METHOD PUBLIC Clone : I_Node
VAR
	pNode : POINTER TO LT_INT;
END_VAR
pNode := __NEW(LT_INT);
Clone := pNode^;
END_METHOD

METHOD PROTECTED OnExecute
VAR
END_VAR
out.Value := in1.Value < in2.Value;
END_METHOD

END_FUNCTION_BLOCK

// Comparison/Nodes/LT/LT_LINT
{attribute 'linkalways'} 
{attribute 'no_explicit_call' := 'This FB is a CLASS and must be accessed using methods or properties'}
{attribute 'enable_dynamic_creation'}
FUNCTION_BLOCK FINAL LT_LINT EXTENDS Node
VAR
	in1 : _LINT(0);
	in2 : _LINT(0);
	out : _BOOL(FALSE);
END_VAR

METHOD FB_init : BOOL
VAR_INPUT
	bInitRetains : BOOL; // if TRUE, the retain variables are initialized (warm start / cold start)
	bInCopyCode : BOOL;  // if TRUE, the instance afterwards gets moved into the copy code (online change)
END_VAR
AddInput('in1',THIS^.in1);
AddInput('in2',THIS^.in2);
AddOutput('out', THIS^.out);
END_METHOD

METHOD PUBLIC Clone : I_Node
VAR
	pNode : POINTER TO LT_LINT;
END_VAR
pNode := __NEW(LT_LINT);
Clone := pNode^;
END_METHOD

METHOD PROTECTED OnExecute
VAR
END_VAR
out.Value := in1.Value < in2.Value;
END_METHOD

END_FUNCTION_BLOCK

// Comparison/Nodes/LT/LT_LREAL
{attribute 'linkalways'} 
{attribute 'no_explicit_call' := 'This FB is a CLASS and must be accessed using methods or properties'}
{attribute 'enable_dynamic_creation'}
FUNCTION_BLOCK FINAL LT_LREAL EXTENDS Node
VAR
	in1 : _LREAL(0.0);
	in2 : _LREAL(0.0);
	out : _BOOL(FALSE);
END_VAR

METHOD FB_init : BOOL
VAR_INPUT
	bInitRetains : BOOL; // if TRUE, the retain variables are initialized (warm start / cold start)
	bInCopyCode : BOOL;  // if TRUE, the instance afterwards gets moved into the copy code (online change)
END_VAR
AddInput('in1',THIS^.in1);
AddInput('in2',THIS^.in2);
AddOutput('out', THIS^.out);
END_METHOD

METHOD PUBLIC Clone : I_Node
VAR
	pNode : POINTER TO LT_LREAL;
END_VAR
pNode := __NEW(LT_LREAL);
Clone := pNode^;
END_METHOD

METHOD PROTECTED OnExecute
VAR
END_VAR
out.Value := in1.Value < in2.Value;
END_METHOD

END_FUNCTION_BLOCK

// Comparison/Nodes/LT/LT_LWORD
{attribute 'linkalways'} 
{attribute 'no_explicit_call' := 'This FB is a CLASS and must be accessed using methods or properties'}
{attribute 'enable_dynamic_creation'}
FUNCTION_BLOCK FINAL LT_LWORD EXTENDS Node
VAR
	in1 : _LWORD(0);
	in2 : _LWORD(0);
	out : _BOOL(FALSE);
END_VAR

METHOD FB_init : BOOL
VAR_INPUT
	bInitRetains : BOOL; // if TRUE, the retain variables are initialized (warm start / cold start)
	bInCopyCode : BOOL;  // if TRUE, the instance afterwards gets moved into the copy code (online change)
END_VAR
AddInput('in1',THIS^.in1);
AddInput('in2',THIS^.in2);
AddOutput('out', THIS^.out);
END_METHOD

METHOD PUBLIC Clone : I_Node
VAR
	pNode : POINTER TO LT_LWORD;
END_VAR
pNode := __NEW(LT_LWORD);
Clone := pNode^;
END_METHOD

METHOD PROTECTED OnExecute
VAR
END_VAR
out.Value := in1.Value < in2.Value;
END_METHOD

END_FUNCTION_BLOCK

// Comparison/Nodes/LT/LT_REAL
{attribute 'linkalways'} 
{attribute 'no_explicit_call' := 'This FB is a CLASS and must be accessed using methods or properties'}
{attribute 'enable_dynamic_creation'}
FUNCTION_BLOCK FINAL LT_REAL EXTENDS Node
VAR
	in1 : _REAL(0.0);
	in2 : _REAL(0.0);
	out : _BOOL(FALSE);
END_VAR

METHOD FB_init : BOOL
VAR_INPUT
	bInitRetains : BOOL; // if TRUE, the retain variables are initialized (warm start / cold start)
	bInCopyCode : BOOL;  // if TRUE, the instance afterwards gets moved into the copy code (online change)
END_VAR
AddInput('in1',THIS^.in1);
AddInput('in2',THIS^.in2);
AddOutput('out', THIS^.out);
END_METHOD

METHOD PUBLIC Clone : I_Node
VAR
	pNode : POINTER TO LT_REAL;
END_VAR
pNode := __NEW(LT_REAL);
Clone := pNode^;
END_METHOD

METHOD PROTECTED OnExecute
VAR
END_VAR
out.Value := in1.Value < in2.Value;
END_METHOD

END_FUNCTION_BLOCK

// Comparison/Nodes/LT/LT_SINT
{attribute 'linkalways'} 
{attribute 'no_explicit_call' := 'This FB is a CLASS and must be accessed using methods or properties'}
{attribute 'enable_dynamic_creation'}
FUNCTION_BLOCK FINAL LT_SINT EXTENDS Node
VAR
	in1 : _SINT(0);
	in2 : _SINT(0);
	out : _BOOL(FALSE);
END_VAR

METHOD FB_init : BOOL
VAR_INPUT
	bInitRetains : BOOL; // if TRUE, the retain variables are initialized (warm start / cold start)
	bInCopyCode : BOOL;  // if TRUE, the instance afterwards gets moved into the copy code (online change)
END_VAR
AddInput('in1',THIS^.in1);
AddInput('in2',THIS^.in2);
AddOutput('out', THIS^.out);
END_METHOD

METHOD PUBLIC Clone : I_Node
VAR
	pNode : POINTER TO LT_SINT;
END_VAR
pNode := __NEW(LT_SINT);
Clone := pNode^;
END_METHOD

METHOD PROTECTED OnExecute
VAR
END_VAR
out.Value := in1.Value < in2.Value;
END_METHOD

END_FUNCTION_BLOCK

// Comparison/Nodes/LT/LT_UDINT
{attribute 'linkalways'} 
{attribute 'no_explicit_call' := 'This FB is a CLASS and must be accessed using methods or properties'}
{attribute 'enable_dynamic_creation'}
FUNCTION_BLOCK FINAL LT_UDINT EXTENDS Node
VAR
	in1 : _UDINT(0);
	in2 : _UDINT(0);
	out : _BOOL(FALSE);
END_VAR

METHOD FB_init : BOOL
VAR_INPUT
	bInitRetains : BOOL; // if TRUE, the retain variables are initialized (warm start / cold start)
	bInCopyCode : BOOL;  // if TRUE, the instance afterwards gets moved into the copy code (online change)
END_VAR
AddInput('in1',THIS^.in1);
AddInput('in2',THIS^.in2);
AddOutput('out', THIS^.out);
END_METHOD

METHOD PUBLIC Clone : I_Node
VAR
	pNode : POINTER TO LT_UDINT;
END_VAR
pNode := __NEW(LT_UDINT);
Clone := pNode^;
END_METHOD

METHOD PROTECTED OnExecute
VAR
END_VAR
out.Value := in1.Value < in2.Value;
END_METHOD

END_FUNCTION_BLOCK

// Comparison/Nodes/LT/LT_UINT
{attribute 'linkalways'} 
{attribute 'no_explicit_call' := 'This FB is a CLASS and must be accessed using methods or properties'}
{attribute 'enable_dynamic_creation'}
FUNCTION_BLOCK FINAL LT_UINT EXTENDS Node
VAR
	in1 : _UINT(0);
	in2 : _UINT(0);
	out : _BOOL(FALSE);
END_VAR

METHOD FB_init : BOOL
VAR_INPUT
	bInitRetains : BOOL; // if TRUE, the retain variables are initialized (warm start / cold start)
	bInCopyCode : BOOL;  // if TRUE, the instance afterwards gets moved into the copy code (online change)
END_VAR
AddInput('in1',THIS^.in1);
AddInput('in2',THIS^.in2);
AddOutput('out', THIS^.out);
END_METHOD

METHOD PUBLIC Clone : I_Node
VAR
	pNode : POINTER TO LT_UINT;
END_VAR
pNode := __NEW(LT_UINT);
Clone := pNode^;
END_METHOD

METHOD PROTECTED OnExecute
VAR
END_VAR
out.Value := in1.Value < in2.Value;
END_METHOD

END_FUNCTION_BLOCK

// Comparison/Nodes/LT/LT_ULINT
{attribute 'linkalways'} 
{attribute 'no_explicit_call' := 'This FB is a CLASS and must be accessed using methods or properties'}
{attribute 'enable_dynamic_creation'}
FUNCTION_BLOCK FINAL LT_ULINT EXTENDS Node
VAR
	in1 : _ULINT(0);
	in2 : _ULINT(0);
	out : _BOOL(FALSE);
END_VAR

METHOD FB_init : BOOL
VAR_INPUT
	bInitRetains : BOOL; // if TRUE, the retain variables are initialized (warm start / cold start)
	bInCopyCode : BOOL;  // if TRUE, the instance afterwards gets moved into the copy code (online change)
END_VAR
AddInput('in1',THIS^.in1);
AddInput('in2',THIS^.in2);
AddOutput('out', THIS^.out);
END_METHOD

METHOD PUBLIC Clone : I_Node
VAR
	pNode : POINTER TO LT_ULINT;
END_VAR
pNode := __NEW(LT_ULINT);
Clone := pNode^;
END_METHOD

METHOD PROTECTED OnExecute
VAR
END_VAR
out.Value := in1.Value < in2.Value;
END_METHOD

END_FUNCTION_BLOCK

// Comparison/Nodes/LT/LT_USINT
{attribute 'linkalways'} 
{attribute 'no_explicit_call' := 'This FB is a CLASS and must be accessed using methods or properties'}
{attribute 'enable_dynamic_creation'}
FUNCTION_BLOCK FINAL LT_USINT EXTENDS Node
VAR
	in1 : _USINT(0);
	in2 : _USINT(0);
	out : _BOOL(FALSE);
END_VAR

METHOD FB_init : BOOL
VAR_INPUT
	bInitRetains : BOOL; // if TRUE, the retain variables are initialized (warm start / cold start)
	bInCopyCode : BOOL;  // if TRUE, the instance afterwards gets moved into the copy code (online change)
END_VAR
AddInput('in1',THIS^.in1);
AddInput('in2',THIS^.in2);
AddOutput('out', THIS^.out);
END_METHOD

METHOD PUBLIC Clone : I_Node
VAR
	pNode : POINTER TO LT_USINT;
END_VAR
pNode := __NEW(LT_USINT);
Clone := pNode^;
END_METHOD

METHOD PROTECTED OnExecute
VAR
END_VAR
out.Value := in1.Value < in2.Value;
END_METHOD

END_FUNCTION_BLOCK

// Comparison/Nodes/LT/LT_WORD
{attribute 'linkalways'} 
{attribute 'no_explicit_call' := 'This FB is a CLASS and must be accessed using methods or properties'}
{attribute 'enable_dynamic_creation'}
FUNCTION_BLOCK FINAL LT_WORD EXTENDS Node
VAR
	in1 : _WORD(0);
	in2 : _WORD(0);
	out : _BOOL(FALSE);
END_VAR

METHOD FB_init : BOOL
VAR_INPUT
	bInitRetains : BOOL; // if TRUE, the retain variables are initialized (warm start / cold start)
	bInCopyCode : BOOL;  // if TRUE, the instance afterwards gets moved into the copy code (online change)
END_VAR
AddInput('in1',THIS^.in1);
AddInput('in2',THIS^.in2);
AddOutput('out', THIS^.out);
END_METHOD

METHOD PUBLIC Clone : I_Node
VAR
	pNode : POINTER TO LT_WORD;
END_VAR
pNode := __NEW(LT_WORD);
Clone := pNode^;
END_METHOD

METHOD PROTECTED OnExecute
VAR
END_VAR
out.Value := in1.Value < in2.Value;
END_METHOD

END_FUNCTION_BLOCK

// Comparison/Nodes/NE/NE_BYTE
{attribute 'linkalways'} 
{attribute 'no_explicit_call' := 'This FB is a CLASS and must be accessed using methods or properties'}
{attribute 'enable_dynamic_creation'}
FUNCTION_BLOCK FINAL NE_BYTE EXTENDS Node
VAR
	in1 : _BYTE(0);
	in2 : _BYTE(0);
	out : _BOOL(FALSE);
END_VAR

METHOD FB_init : BOOL
VAR_INPUT
	bInitRetains : BOOL; // if TRUE, the retain variables are initialized (warm start / cold start)
	bInCopyCode : BOOL;  // if TRUE, the instance afterwards gets moved into the copy code (online change)
END_VAR
AddInput('in1',THIS^.in1);
AddInput('in2',THIS^.in2);
AddOutput('out', THIS^.out);
END_METHOD

METHOD PUBLIC Clone : I_Node
VAR
	pNode : POINTER TO NE_BYTE;
END_VAR
pNode := __NEW(NE_BYTE);
Clone := pNode^;
END_METHOD

METHOD PROTECTED OnExecute
VAR
END_VAR
out.Value := in1.Value <> in2.Value;
END_METHOD

END_FUNCTION_BLOCK

// Comparison/Nodes/NE/NE_DINT
{attribute 'linkalways'} 
{attribute 'no_explicit_call' := 'This FB is a CLASS and must be accessed using methods or properties'}
{attribute 'enable_dynamic_creation'}
FUNCTION_BLOCK FINAL NE_DINT EXTENDS Node
VAR
	in1 : _DINT(0);
	in2 : _DINT(0);
	out : _BOOL(FALSE);
END_VAR

METHOD FB_init : BOOL
VAR_INPUT
	bInitRetains : BOOL; // if TRUE, the retain variables are initialized (warm start / cold start)
	bInCopyCode : BOOL;  // if TRUE, the instance afterwards gets moved into the copy code (online change)
END_VAR
AddInput('in1',THIS^.in1);
AddInput('in2',THIS^.in2);
AddOutput('out', THIS^.out);
END_METHOD

METHOD PUBLIC Clone : I_Node
VAR
	pNode : POINTER TO NE_DINT;
END_VAR
pNode := __NEW(NE_DINT);
Clone := pNode^;
END_METHOD

METHOD PROTECTED OnExecute
VAR
END_VAR
out.Value := in1.Value <> in2.Value;
END_METHOD

END_FUNCTION_BLOCK

// Comparison/Nodes/NE/NE_DWORD
{attribute 'linkalways'} 
{attribute 'no_explicit_call' := 'This FB is a CLASS and must be accessed using methods or properties'}
{attribute 'enable_dynamic_creation'}
FUNCTION_BLOCK FINAL NE_DWORD EXTENDS Node
VAR
	in1 : _DWORD(0);
	in2 : _DWORD(0);
	out : _BOOL(FALSE);
END_VAR

METHOD FB_init : BOOL
VAR_INPUT
	bInitRetains : BOOL; // if TRUE, the retain variables are initialized (warm start / cold start)
	bInCopyCode : BOOL;  // if TRUE, the instance afterwards gets moved into the copy code (online change)
END_VAR
AddInput('in1',THIS^.in1);
AddInput('in2',THIS^.in2);
AddOutput('out', THIS^.out);
END_METHOD

METHOD PUBLIC Clone : I_Node
VAR
	pNode : POINTER TO NE_DWORD;
END_VAR
pNode := __NEW(NE_DWORD);
Clone := pNode^;
END_METHOD

METHOD PROTECTED OnExecute
VAR
END_VAR
out.Value := in1.Value <> in2.Value;
END_METHOD

END_FUNCTION_BLOCK

// Comparison/Nodes/NE/NE_INT
{attribute 'linkalways'} 
{attribute 'no_explicit_call' := 'This FB is a CLASS and must be accessed using methods or properties'}
{attribute 'enable_dynamic_creation'}
FUNCTION_BLOCK FINAL NE_INT EXTENDS Node
VAR
	in1 : _INT(0);
	in2 : _INT(0);
	out : _BOOL(FALSE);
END_VAR

METHOD FB_init : BOOL
VAR_INPUT
	bInitRetains : BOOL; // if TRUE, the retain variables are initialized (warm start / cold start)
	bInCopyCode : BOOL;  // if TRUE, the instance afterwards gets moved into the copy code (online change)
END_VAR
AddInput('in1',THIS^.in1);
AddInput('in2',THIS^.in2);
AddOutput('out', THIS^.out);
END_METHOD

METHOD PUBLIC Clone : I_Node
VAR
	pNode : POINTER TO NE_INT;
END_VAR
pNode := __NEW(NE_INT);
Clone := pNode^;
END_METHOD

METHOD PROTECTED OnExecute
VAR
END_VAR
out.Value := in1.Value <> in2.Value;
END_METHOD

END_FUNCTION_BLOCK

// Comparison/Nodes/NE/NE_LINT
{attribute 'linkalways'} 
{attribute 'no_explicit_call' := 'This FB is a CLASS and must be accessed using methods or properties'}
{attribute 'enable_dynamic_creation'}
FUNCTION_BLOCK FINAL NE_LINT EXTENDS Node
VAR
	in1 : _LINT(0);
	in2 : _LINT(0);
	out : _BOOL(FALSE);
END_VAR

METHOD FB_init : BOOL
VAR_INPUT
	bInitRetains : BOOL; // if TRUE, the retain variables are initialized (warm start / cold start)
	bInCopyCode : BOOL;  // if TRUE, the instance afterwards gets moved into the copy code (online change)
END_VAR
AddInput('in1',THIS^.in1);
AddInput('in2',THIS^.in2);
AddOutput('out', THIS^.out);
END_METHOD

METHOD PUBLIC Clone : I_Node
VAR
	pNode : POINTER TO NE_LINT;
END_VAR
pNode := __NEW(NE_LINT);
Clone := pNode^;
END_METHOD

METHOD PROTECTED OnExecute
VAR
END_VAR
out.Value := in1.Value <> in2.Value;
END_METHOD

END_FUNCTION_BLOCK

// Comparison/Nodes/NE/NE_LREAL
{attribute 'linkalways'} 
{attribute 'no_explicit_call' := 'This FB is a CLASS and must be accessed using methods or properties'}
{attribute 'enable_dynamic_creation'}
FUNCTION_BLOCK FINAL NE_LREAL EXTENDS Node
VAR
	in1 : _LREAL(0.0);
	in2 : _LREAL(0.0);
	out : _BOOL(FALSE);
END_VAR

METHOD FB_init : BOOL
VAR_INPUT
	bInitRetains : BOOL; // if TRUE, the retain variables are initialized (warm start / cold start)
	bInCopyCode : BOOL;  // if TRUE, the instance afterwards gets moved into the copy code (online change)
END_VAR
AddInput('in1',THIS^.in1);
AddInput('in2',THIS^.in2);
AddOutput('out', THIS^.out);
END_METHOD

METHOD PUBLIC Clone : I_Node
VAR
	pNode : POINTER TO NE_LREAL;
END_VAR
pNode := __NEW(NE_LREAL);
Clone := pNode^;
END_METHOD

METHOD PROTECTED OnExecute
VAR
END_VAR
out.Value := in1.Value <> in2.Value;
END_METHOD

END_FUNCTION_BLOCK

// Comparison/Nodes/NE/NE_LWORD
{attribute 'linkalways'} 
{attribute 'no_explicit_call' := 'This FB is a CLASS and must be accessed using methods or properties'}
{attribute 'enable_dynamic_creation'}
FUNCTION_BLOCK FINAL NE_LWORD EXTENDS Node
VAR
	in1 : _LWORD(0);
	in2 : _LWORD(0);
	out : _BOOL(FALSE);
END_VAR

METHOD FB_init : BOOL
VAR_INPUT
	bInitRetains : BOOL; // if TRUE, the retain variables are initialized (warm start / cold start)
	bInCopyCode : BOOL;  // if TRUE, the instance afterwards gets moved into the copy code (online change)
END_VAR
AddInput('in1',THIS^.in1);
AddInput('in2',THIS^.in2);
AddOutput('out', THIS^.out);
END_METHOD

METHOD PUBLIC Clone : I_Node
VAR
	pNode : POINTER TO NE_LWORD;
END_VAR
pNode := __NEW(NE_LWORD);
Clone := pNode^;
END_METHOD

METHOD PROTECTED OnExecute
VAR
END_VAR
out.Value := in1.Value <> in2.Value;
END_METHOD

END_FUNCTION_BLOCK

// Comparison/Nodes/NE/NE_REAL
{attribute 'linkalways'} 
{attribute 'no_explicit_call' := 'This FB is a CLASS and must be accessed using methods or properties'}
{attribute 'enable_dynamic_creation'}
FUNCTION_BLOCK FINAL NE_REAL EXTENDS Node
VAR
	in1 : _REAL(0.0);
	in2 : _REAL(0.0);
	out : _BOOL(FALSE);
END_VAR

METHOD FB_init : BOOL
VAR_INPUT
	bInitRetains : BOOL; // if TRUE, the retain variables are initialized (warm start / cold start)
	bInCopyCode : BOOL;  // if TRUE, the instance afterwards gets moved into the copy code (online change)
END_VAR
AddInput('in1',THIS^.in1);
AddInput('in2',THIS^.in2);
AddOutput('out', THIS^.out);
END_METHOD

METHOD PUBLIC Clone : I_Node
VAR
	pNode : POINTER TO NE_REAL;
END_VAR
pNode := __NEW(NE_REAL);
Clone := pNode^;
END_METHOD

METHOD PROTECTED OnExecute
VAR
END_VAR
out.Value := in1.Value <> in2.Value;
END_METHOD

END_FUNCTION_BLOCK

// Comparison/Nodes/NE/NE_SINT
{attribute 'linkalways'} 
{attribute 'no_explicit_call' := 'This FB is a CLASS and must be accessed using methods or properties'}
{attribute 'enable_dynamic_creation'}
FUNCTION_BLOCK FINAL NE_SINT EXTENDS Node
VAR
	in1 : _SINT(0);
	in2 : _SINT(0);
	out : _BOOL(FALSE);
END_VAR

METHOD FB_init : BOOL
VAR_INPUT
	bInitRetains : BOOL; // if TRUE, the retain variables are initialized (warm start / cold start)
	bInCopyCode : BOOL;  // if TRUE, the instance afterwards gets moved into the copy code (online change)
END_VAR
AddInput('in1',THIS^.in1);
AddInput('in2',THIS^.in2);
AddOutput('out', THIS^.out);
END_METHOD

METHOD PUBLIC Clone : I_Node
VAR
	pNode : POINTER TO NE_SINT;
END_VAR
pNode := __NEW(NE_SINT);
Clone := pNode^;
END_METHOD

METHOD PROTECTED OnExecute
VAR
END_VAR
out.Value := in1.Value <> in2.Value;
END_METHOD

END_FUNCTION_BLOCK

// Comparison/Nodes/NE/NE_UDINT
{attribute 'linkalways'} 
{attribute 'no_explicit_call' := 'This FB is a CLASS and must be accessed using methods or properties'}
{attribute 'enable_dynamic_creation'}
FUNCTION_BLOCK FINAL NE_UDINT EXTENDS Node
VAR
	in1 : _UDINT(0);
	in2 : _UDINT(0);
	out : _BOOL(FALSE);
END_VAR

METHOD FB_init : BOOL
VAR_INPUT
	bInitRetains : BOOL; // if TRUE, the retain variables are initialized (warm start / cold start)
	bInCopyCode : BOOL;  // if TRUE, the instance afterwards gets moved into the copy code (online change)
END_VAR
AddInput('in1',THIS^.in1);
AddInput('in2',THIS^.in2);
AddOutput('out', THIS^.out);
END_METHOD

METHOD PUBLIC Clone : I_Node
VAR
	pNode : POINTER TO NE_UDINT;
END_VAR
pNode := __NEW(NE_UDINT);
Clone := pNode^;
END_METHOD

METHOD PROTECTED OnExecute
VAR
END_VAR
out.Value := in1.Value <> in2.Value;
END_METHOD

END_FUNCTION_BLOCK

// Comparison/Nodes/NE/NE_UINT
{attribute 'linkalways'} 
{attribute 'no_explicit_call' := 'This FB is a CLASS and must be accessed using methods or properties'}
{attribute 'enable_dynamic_creation'}
FUNCTION_BLOCK FINAL NE_UINT EXTENDS Node
VAR
	in1 : _UINT(0);
	in2 : _UINT(0);
	out : _BOOL(FALSE);
END_VAR

METHOD FB_init : BOOL
VAR_INPUT
	bInitRetains : BOOL; // if TRUE, the retain variables are initialized (warm start / cold start)
	bInCopyCode : BOOL;  // if TRUE, the instance afterwards gets moved into the copy code (online change)
END_VAR
AddInput('in1',THIS^.in1);
AddInput('in2',THIS^.in2);
AddOutput('out', THIS^.out);
END_METHOD

METHOD PUBLIC Clone : I_Node
VAR
	pNode : POINTER TO NE_UINT;
END_VAR
pNode := __NEW(NE_UINT);
Clone := pNode^;
END_METHOD

METHOD PROTECTED OnExecute
VAR
END_VAR
out.Value := in1.Value <> in2.Value;
END_METHOD

END_FUNCTION_BLOCK

// Comparison/Nodes/NE/NE_ULINT
{attribute 'linkalways'} 
{attribute 'no_explicit_call' := 'This FB is a CLASS and must be accessed using methods or properties'}
{attribute 'enable_dynamic_creation'}
FUNCTION_BLOCK FINAL NE_ULINT EXTENDS Node
VAR
	in1 : _ULINT(0);
	in2 : _ULINT(0);
	out : _BOOL(FALSE);
END_VAR

METHOD FB_init : BOOL
VAR_INPUT
	bInitRetains : BOOL; // if TRUE, the retain variables are initialized (warm start / cold start)
	bInCopyCode : BOOL;  // if TRUE, the instance afterwards gets moved into the copy code (online change)
END_VAR
AddInput('in1',THIS^.in1);
AddInput('in2',THIS^.in2);
AddOutput('out', THIS^.out);
END_METHOD

METHOD PUBLIC Clone : I_Node
VAR
	pNode : POINTER TO NE_ULINT;
END_VAR
pNode := __NEW(NE_ULINT);
Clone := pNode^;
END_METHOD

METHOD PROTECTED OnExecute
VAR
END_VAR
out.Value := in1.Value <> in2.Value;
END_METHOD

END_FUNCTION_BLOCK

// Comparison/Nodes/NE/NE_USINT
{attribute 'linkalways'} 
{attribute 'no_explicit_call' := 'This FB is a CLASS and must be accessed using methods or properties'}
{attribute 'enable_dynamic_creation'}
FUNCTION_BLOCK FINAL NE_USINT EXTENDS Node
VAR
	in1 : _USINT(0);
	in2 : _USINT(0);
	out : _BOOL(FALSE);
END_VAR

METHOD FB_init : BOOL
VAR_INPUT
	bInitRetains : BOOL; // if TRUE, the retain variables are initialized (warm start / cold start)
	bInCopyCode : BOOL;  // if TRUE, the instance afterwards gets moved into the copy code (online change)
END_VAR
AddInput('in1',THIS^.in1);
AddInput('in2',THIS^.in2);
AddOutput('out', THIS^.out);
END_METHOD

METHOD PUBLIC Clone : I_Node
VAR
	pNode : POINTER TO NE_USINT;
END_VAR
pNode := __NEW(NE_USINT);
Clone := pNode^;
END_METHOD

METHOD PROTECTED OnExecute
VAR
END_VAR
out.Value := in1.Value <> in2.Value;
END_METHOD

END_FUNCTION_BLOCK

// Comparison/Nodes/NE/NE_WORD
{attribute 'linkalways'} 
{attribute 'no_explicit_call' := 'This FB is a CLASS and must be accessed using methods or properties'}
{attribute 'enable_dynamic_creation'}
FUNCTION_BLOCK FINAL NE_WORD EXTENDS Node
VAR
	in1 : _WORD(0);
	in2 : _WORD(0);
	out : _BOOL(FALSE);
END_VAR

METHOD FB_init : BOOL
VAR_INPUT
	bInitRetains : BOOL; // if TRUE, the retain variables are initialized (warm start / cold start)
	bInCopyCode : BOOL;  // if TRUE, the instance afterwards gets moved into the copy code (online change)
END_VAR
AddInput('in1',THIS^.in1);
AddInput('in2',THIS^.in2);
AddOutput('out', THIS^.out);
END_METHOD

METHOD PUBLIC Clone : I_Node
VAR
	pNode : POINTER TO NE_WORD;
END_VAR
pNode := __NEW(NE_WORD);
Clone := pNode^;
END_METHOD

METHOD PROTECTED OnExecute
VAR
END_VAR
out.Value := in1.Value <> in2.Value;
END_METHOD

END_FUNCTION_BLOCK

// Comparison/MathComparisonPack
{attribute 'linkalways'} 
{attribute 'no_explicit_call' := 'This FB is a CLASS and must be accessed using methods or properties'}
{attribute 'enable_dynamic_creation'}
FUNCTION_BLOCK MathComparisonPack IMPLEMENTS I_GraphPack
VAR
	GT_BYTE : GT_BYTE;
	GT_DINT : GT_DINT;
	GT_DWORD : GT_DWORD;
	GT_INT : GT_INT;
	GT_LINT : GT_LINT;
	GT_LREAL : GT_LREAL;
	GT_LWORD : GT_LWORD;
	GT_REAL : GT_REAL;
	GT_SINT : GT_SINT;
	GT_UDINT : GT_UDINT;
	GT_UINT : GT_UINT;
	GT_ULINT : GT_ULINT;
	GT_USINT : GT_USINT;
	GT_WORD : GT_WORD;
	
	LT_BYTE : LT_BYTE;
	LT_DINT : LT_DINT;
	LT_DWORD : LT_DWORD;
	LT_INT : LT_INT;
	LT_LINT : LT_LINT;
	LT_LREAL : LT_LREAL;
	LT_LWORD : LT_LWORD;
	LT_REAL : LT_REAL;
	LT_SINT : LT_SINT;
	LT_UDINT : LT_UDINT;
	LT_UINT : LT_UINT;
	LT_ULINT : LT_ULINT;
	LT_USINT : LT_USINT;
	LT_WORD : LT_WORD;
	
	EQ_BYTE : EQ_BYTE;
	EQ_DINT : EQ_DINT;
	EQ_DWORD : EQ_DWORD;
	EQ_INT : EQ_INT;
	EQ_LINT : EQ_LINT;
	EQ_LREAL : EQ_LREAL;
	EQ_LWORD : EQ_LWORD;
	EQ_REAL : EQ_REAL;
	EQ_SINT : EQ_SINT;
	EQ_UDINT : EQ_UDINT;
	EQ_UINT : EQ_UINT;
	EQ_ULINT : EQ_ULINT;
	EQ_USINT : EQ_USINT;
	EQ_WORD : EQ_WORD;
	
	NE_BYTE : NE_BYTE;
	NE_DINT : NE_DINT;
	NE_DWORD : NE_DWORD;
	NE_INT : NE_INT;
	NE_LINT : NE_LINT;
	NE_LREAL : NE_LREAL;
	NE_LWORD : NE_LWORD;
	NE_REAL : NE_REAL;
	NE_SINT : NE_SINT;
	NE_UDINT : NE_UDINT;
	NE_UINT : NE_UINT;
	NE_ULINT : NE_ULINT;
	NE_USINT : NE_USINT;
	NE_WORD : NE_WORD;
	
	LE_BYTE : LE_BYTE;
	LE_DINT : LE_DINT;
	LE_DWORD : LE_DWORD;
	LE_INT : LE_INT;
	LE_LINT : LE_LINT;
	LE_LREAL : LE_LREAL;
	LE_LWORD : LE_LWORD;
	LE_REAL : LE_REAL;
	LE_SINT : LE_SINT;
	LE_UDINT : LE_UDINT;
	LE_UINT : LE_UINT;
	LE_ULINT : LE_ULINT;
	LE_USINT : LE_USINT;
	LE_WORD : LE_WORD;
	
	GE_BYTE : GE_BYTE;
	GE_DINT : GE_DINT;
	GE_DWORD : GE_DWORD;
	GE_INT : GE_INT;
	GE_LINT : GE_LINT;
	GE_LREAL : GE_LREAL;
	GE_LWORD : GE_LWORD;
	GE_REAL : GE_REAL;
	GE_SINT : GE_SINT;
	GE_UDINT : GE_UDINT;
	GE_UINT : GE_UINT;
	GE_ULINT : GE_ULINT;
	GE_USINT : GE_USINT;
	GE_WORD : GE_WORD;
END_VAR

METHOD Register
VAR_INPUT
	Datatypes : I_Datatypes;
	NodeFactory : I_NodeFactory;
END_VAR
NodeFactory.AddNodeAsPrototype('Math/Comparison/GT/GT_BYTE',GT_BYTE);
NodeFactory.AddNodeAsPrototype('Math/Comparison/GT/GT_DINT',GT_DINT);
NodeFactory.AddNodeAsPrototype('Math/Comparison/GT/GT_DWORD',GT_DWORD);
NodeFactory.AddNodeAsPrototype('Math/Comparison/GT/GT_INT',GT_INT);
NodeFactory.AddNodeAsPrototype('Math/Comparison/GT/GT_LINT',GT_LINT);
NodeFactory.AddNodeAsPrototype('Math/Comparison/GT/GT_LREAL',GT_LREAL);
NodeFactory.AddNodeAsPrototype('Math/Comparison/GT/GT_LWORD',GT_LWORD);
NodeFactory.AddNodeAsPrototype('Math/Comparison/GT/GT_REAL',GT_REAL);
NodeFactory.AddNodeAsPrototype('Math/Comparison/GT/GT_SINT',GT_SINT);
NodeFactory.AddNodeAsPrototype('Math/Comparison/GT/GT_UDINT',GT_UDINT);
NodeFactory.AddNodeAsPrototype('Math/Comparison/GT/GT_UINT',GT_UINT);
NodeFactory.AddNodeAsPrototype('Math/Comparison/GT/GT_ULINT',GT_ULINT);
NodeFactory.AddNodeAsPrototype('Math/Comparison/GT/GT_USINT',GT_USINT);
NodeFactory.AddNodeAsPrototype('Math/Comparison/GT/GT_WORD',GT_WORD);

NodeFactory.AddNodeAsPrototype('Math/Comparison/LT/LT_BYTE',LT_BYTE);
NodeFactory.AddNodeAsPrototype('Math/Comparison/LT/LT_DINT',LT_DINT);
NodeFactory.AddNodeAsPrototype('Math/Comparison/LT/LT_DWORD',LT_DWORD);
NodeFactory.AddNodeAsPrototype('Math/Comparison/LT/LT_INT',LT_INT);
NodeFactory.AddNodeAsPrototype('Math/Comparison/LT/LT_LINT',LT_LINT);
NodeFactory.AddNodeAsPrototype('Math/Comparison/LT/LT_LREAL',LT_LREAL);
NodeFactory.AddNodeAsPrototype('Math/Comparison/LT/LT_LWORD',LT_LWORD);
NodeFactory.AddNodeAsPrototype('Math/Comparison/LT/LT_REAL',LT_REAL);
NodeFactory.AddNodeAsPrototype('Math/Comparison/LT/LT_SINT',LT_SINT);
NodeFactory.AddNodeAsPrototype('Math/Comparison/LT/LT_UDINT',LT_UDINT);
NodeFactory.AddNodeAsPrototype('Math/Comparison/LT/LT_UINT',LT_UINT);
NodeFactory.AddNodeAsPrototype('Math/Comparison/LT/LT_ULINT',LT_ULINT);
NodeFactory.AddNodeAsPrototype('Math/Comparison/LT/LT_USINT',LT_USINT);
NodeFactory.AddNodeAsPrototype('Math/Comparison/LT/LT_WORD',LT_WORD);

NodeFactory.AddNodeAsPrototype('Math/Comparison/EQ/EQ_BYTE',EQ_BYTE);
NodeFactory.AddNodeAsPrototype('Math/Comparison/EQ/EQ_DINT',EQ_DINT);
NodeFactory.AddNodeAsPrototype('Math/Comparison/EQ/EQ_DWORD',EQ_DWORD);
NodeFactory.AddNodeAsPrototype('Math/Comparison/EQ/EQ_INT',EQ_INT);
NodeFactory.AddNodeAsPrototype('Math/Comparison/EQ/EQ_LINT',EQ_LINT);
NodeFactory.AddNodeAsPrototype('Math/Comparison/EQ/EQ_LREAL',EQ_LREAL);
NodeFactory.AddNodeAsPrototype('Math/Comparison/EQ/EQ_LWORD',EQ_LWORD);
NodeFactory.AddNodeAsPrototype('Math/Comparison/EQ/EQ_REAL',EQ_REAL);
NodeFactory.AddNodeAsPrototype('Math/Comparison/EQ/EQ_SINT',EQ_SINT);
NodeFactory.AddNodeAsPrototype('Math/Comparison/EQ/EQ_UDINT',EQ_UDINT);
NodeFactory.AddNodeAsPrototype('Math/Comparison/EQ/EQ_UINT',EQ_UINT);
NodeFactory.AddNodeAsPrototype('Math/Comparison/EQ/EQ_ULINT',EQ_ULINT);
NodeFactory.AddNodeAsPrototype('Math/Comparison/EQ/EQ_USINT',EQ_USINT);
NodeFactory.AddNodeAsPrototype('Math/Comparison/EQ/EQ_WORD',EQ_WORD);

NodeFactory.AddNodeAsPrototype('Math/Comparison/NE/NE_BYTE',NE_BYTE);
NodeFactory.AddNodeAsPrototype('Math/Comparison/NE/NE_DINT',NE_DINT);
NodeFactory.AddNodeAsPrototype('Math/Comparison/NE/NE_DWORD',NE_DWORD);
NodeFactory.AddNodeAsPrototype('Math/Comparison/NE/NE_INT',NE_INT);
NodeFactory.AddNodeAsPrototype('Math/Comparison/NE/NE_LINT',NE_LINT);
NodeFactory.AddNodeAsPrototype('Math/Comparison/NE/NE_LREAL',NE_LREAL);
NodeFactory.AddNodeAsPrototype('Math/Comparison/NE/NE_LWORD',NE_LWORD);
NodeFactory.AddNodeAsPrototype('Math/Comparison/NE/NE_REAL',NE_REAL);
NodeFactory.AddNodeAsPrototype('Math/Comparison/NE/NE_SINT',NE_SINT);
NodeFactory.AddNodeAsPrototype('Math/Comparison/NE/NE_UDINT',NE_UDINT);
NodeFactory.AddNodeAsPrototype('Math/Comparison/NE/NE_UINT',NE_UINT);
NodeFactory.AddNodeAsPrototype('Math/Comparison/NE/NE_ULINT',NE_ULINT);
NodeFactory.AddNodeAsPrototype('Math/Comparison/NE/NE_USINT',NE_USINT);
NodeFactory.AddNodeAsPrototype('Math/Comparison/NE/NE_WORD',NE_WORD);

NodeFactory.AddNodeAsPrototype('Math/Comparison/LE/LE_BYTE',LE_BYTE);
NodeFactory.AddNodeAsPrototype('Math/Comparison/LE/LE_DINT',LE_DINT);
NodeFactory.AddNodeAsPrototype('Math/Comparison/LE/LE_DWORD',LE_DWORD);
NodeFactory.AddNodeAsPrototype('Math/Comparison/LE/LE_INT',LE_INT);
NodeFactory.AddNodeAsPrototype('Math/Comparison/LE/LE_LINT',LE_LINT);
NodeFactory.AddNodeAsPrototype('Math/Comparison/LE/LE_LREAL',LE_LREAL);
NodeFactory.AddNodeAsPrototype('Math/Comparison/LE/LE_LWORD',LE_LWORD);
NodeFactory.AddNodeAsPrototype('Math/Comparison/LE/LE_REAL',LE_REAL);
NodeFactory.AddNodeAsPrototype('Math/Comparison/LE/LE_SINT',LE_SINT);
NodeFactory.AddNodeAsPrototype('Math/Comparison/LE/LE_UDINT',LE_UDINT);
NodeFactory.AddNodeAsPrototype('Math/Comparison/LE/LE_UINT',LE_UINT);
NodeFactory.AddNodeAsPrototype('Math/Comparison/LE/LE_ULINT',LE_ULINT);
NodeFactory.AddNodeAsPrototype('Math/Comparison/LE/LE_USINT',LE_USINT);
NodeFactory.AddNodeAsPrototype('Math/Comparison/LE/LE_WORD',LE_WORD);

NodeFactory.AddNodeAsPrototype('Math/Comparison/GE/GE_BYTE',GE_BYTE);
NodeFactory.AddNodeAsPrototype('Math/Comparison/GE/GE_DINT',GE_DINT);
NodeFactory.AddNodeAsPrototype('Math/Comparison/GE/GE_DWORD',GE_DWORD);
NodeFactory.AddNodeAsPrototype('Math/Comparison/GE/GE_INT',GE_INT);
NodeFactory.AddNodeAsPrototype('Math/Comparison/GE/GE_LINT',GE_LINT);
NodeFactory.AddNodeAsPrototype('Math/Comparison/GE/GE_LREAL',GE_LREAL);
NodeFactory.AddNodeAsPrototype('Math/Comparison/GE/GE_LWORD',GE_LWORD);
NodeFactory.AddNodeAsPrototype('Math/Comparison/GE/GE_REAL',GE_REAL);
NodeFactory.AddNodeAsPrototype('Math/Comparison/GE/GE_SINT',GE_SINT);
NodeFactory.AddNodeAsPrototype('Math/Comparison/GE/GE_UDINT',GE_UDINT);
NodeFactory.AddNodeAsPrototype('Math/Comparison/GE/GE_UINT',GE_UINT);
NodeFactory.AddNodeAsPrototype('Math/Comparison/GE/GE_ULINT',GE_ULINT);
NodeFactory.AddNodeAsPrototype('Math/Comparison/GE/GE_USINT',GE_USINT);
NodeFactory.AddNodeAsPrototype('Math/Comparison/GE/GE_WORD',GE_WORD);
END_METHOD

END_FUNCTION_BLOCK

// Core/Nodes/ADD/ADD_BYTE
{attribute 'linkalways'} 
{attribute 'no_explicit_call' := 'This FB is a CLASS and must be accessed using methods or properties'}
{attribute 'enable_dynamic_creation'}
FUNCTION_BLOCK FINAL ADD_BYTE EXTENDS Node
VAR
	in1 : _BYTE(0);
	in2 : _BYTE(0);
	out : _BYTE(0);
END_VAR

METHOD FB_init : BOOL
VAR_INPUT
	bInitRetains : BOOL; // if TRUE, the retain variables are initialized (warm start / cold start)
	bInCopyCode : BOOL;  // if TRUE, the instance afterwards gets moved into the copy code (online change)
END_VAR
AddInput('in1',THIS^.in1);
AddInput('in2',THIS^.in2);
AddOutput('out', THIS^.out);
END_METHOD

METHOD PUBLIC Clone : I_Node
VAR
	pNode : POINTER TO ADD_BYTE;
END_VAR
pNode := __NEW(ADD_BYTE);
Clone := pNode^;
END_METHOD

METHOD PROTECTED OnExecute
VAR
END_VAR
out.Value := in1.Value + in2.Value;
END_METHOD

END_FUNCTION_BLOCK

// Core/Nodes/ADD/ADD_DINT
{attribute 'linkalways'} 
{attribute 'no_explicit_call' := 'This FB is a CLASS and must be accessed using methods or properties'}
{attribute 'enable_dynamic_creation'}
FUNCTION_BLOCK FINAL ADD_DINT EXTENDS Node
VAR
	in1 : _DINT(0);
	in2 : _DINT(0);
	out : _DINT(0);
END_VAR

METHOD FB_init : BOOL
VAR_INPUT
	bInitRetains : BOOL; // if TRUE, the retain variables are initialized (warm start / cold start)
	bInCopyCode : BOOL;  // if TRUE, the instance afterwards gets moved into the copy code (online change)
END_VAR
AddInput('in1',THIS^.in1);
AddInput('in2',THIS^.in2);
AddOutput('out', THIS^.out);
END_METHOD

METHOD PUBLIC Clone : I_Node
VAR
	pNode : POINTER TO ADD_DINT;
END_VAR
pNode := __NEW(ADD_DINT);
Clone := pNode^;
END_METHOD

METHOD PROTECTED OnExecute
VAR
END_VAR
out.Value := in1.Value + in2.Value;
END_METHOD

END_FUNCTION_BLOCK

// Core/Nodes/ADD/ADD_DWORD
{attribute 'linkalways'} 
{attribute 'no_explicit_call' := 'This FB is a CLASS and must be accessed using methods or properties'}
{attribute 'enable_dynamic_creation'}
FUNCTION_BLOCK FINAL ADD_DWORD EXTENDS Node
VAR
	in1 : _DWORD(0);
	in2 : _DWORD(0);
	out : _DWORD(0);
END_VAR

METHOD FB_init : BOOL
VAR_INPUT
	bInitRetains : BOOL; // if TRUE, the retain variables are initialized (warm start / cold start)
	bInCopyCode : BOOL;  // if TRUE, the instance afterwards gets moved into the copy code (online change)
END_VAR
AddInput('in1',THIS^.in1);
AddInput('in2',THIS^.in2);
AddOutput('out', THIS^.out);
END_METHOD

METHOD PUBLIC Clone : I_Node
VAR
	pNode : POINTER TO ADD_DWORD;
END_VAR
pNode := __NEW(ADD_DWORD);
Clone := pNode^;
END_METHOD

METHOD PROTECTED OnExecute
VAR
END_VAR
out.Value := in1.Value + in2.Value;
END_METHOD

END_FUNCTION_BLOCK

// Core/Nodes/ADD/ADD_INT
{attribute 'linkalways'} 
{attribute 'no_explicit_call' := 'This FB is a CLASS and must be accessed using methods or properties'}
{attribute 'enable_dynamic_creation'}
FUNCTION_BLOCK FINAL ADD_INT EXTENDS Node
VAR
	in1 : _INT(0);
	in2 : _INT(0);
	out : _INT(0);
END_VAR

METHOD FB_init : BOOL
VAR_INPUT
	bInitRetains : BOOL; // if TRUE, the retain variables are initialized (warm start / cold start)
	bInCopyCode : BOOL;  // if TRUE, the instance afterwards gets moved into the copy code (online change)
END_VAR
AddInput('in1',THIS^.in1);
AddInput('in2',THIS^.in2);
AddOutput('out', THIS^.out);
END_METHOD

METHOD PUBLIC Clone : I_Node
VAR
	pNode : POINTER TO ADD_INT;
END_VAR
pNode := __NEW(ADD_INT);
Clone := pNode^;
END_METHOD

METHOD PROTECTED OnExecute
VAR
END_VAR
out.Value := in1.Value + in2.Value;
END_METHOD

END_FUNCTION_BLOCK

// Core/Nodes/ADD/ADD_LINT
{attribute 'linkalways'} 
{attribute 'no_explicit_call' := 'This FB is a CLASS and must be accessed using methods or properties'}
{attribute 'enable_dynamic_creation'}
FUNCTION_BLOCK FINAL ADD_LINT EXTENDS Node
VAR
	in1 : _LINT(0);
	in2 : _LINT(0);
	out : _LINT(0);
END_VAR

METHOD FB_init : BOOL
VAR_INPUT
	bInitRetains : BOOL; // if TRUE, the retain variables are initialized (warm start / cold start)
	bInCopyCode : BOOL;  // if TRUE, the instance afterwards gets moved into the copy code (online change)
END_VAR
AddInput('in1',THIS^.in1);
AddInput('in2',THIS^.in2);
AddOutput('out', THIS^.out);
END_METHOD

METHOD PUBLIC Clone : I_Node
VAR
	pNode : POINTER TO ADD_LINT;
END_VAR
pNode := __NEW(ADD_LINT);
Clone := pNode^;
END_METHOD

METHOD PROTECTED OnExecute
VAR
END_VAR
out.Value := in1.Value + in2.Value;
END_METHOD

END_FUNCTION_BLOCK

// Core/Nodes/ADD/ADD_LREAL
{attribute 'linkalways'} 
{attribute 'no_explicit_call' := 'This FB is a CLASS and must be accessed using methods or properties'}
{attribute 'enable_dynamic_creation'}
FUNCTION_BLOCK FINAL ADD_LREAL EXTENDS Node
VAR
	in1 : _LREAL(0.0);
	in2 : _LREAL(0.0);
	out : _LREAL(0.0);
END_VAR

METHOD FB_init : BOOL
VAR_INPUT
	bInitRetains : BOOL; // if TRUE, the retain variables are initialized (warm start / cold start)
	bInCopyCode : BOOL;  // if TRUE, the instance afterwards gets moved into the copy code (online change)
END_VAR
AddInput('in1',THIS^.in1);
AddInput('in2',THIS^.in2);
AddOutput('out', THIS^.out);
END_METHOD

METHOD PUBLIC Clone : I_Node
VAR
	pNode : POINTER TO ADD_LREAL;
END_VAR
pNode := __NEW(ADD_LREAL);
Clone := pNode^;
END_METHOD

METHOD PROTECTED OnExecute
VAR
END_VAR
out.Value := in1.Value + in2.Value;
END_METHOD

END_FUNCTION_BLOCK

// Core/Nodes/ADD/ADD_LWORD
{attribute 'linkalways'} 
{attribute 'no_explicit_call' := 'This FB is a CLASS and must be accessed using methods or properties'}
{attribute 'enable_dynamic_creation'}
FUNCTION_BLOCK FINAL ADD_LWORD EXTENDS Node
VAR
	in1 : _LWORD(0);
	in2 : _LWORD(0);
	out : _LWORD(0);
END_VAR

METHOD FB_init : BOOL
VAR_INPUT
	bInitRetains : BOOL; // if TRUE, the retain variables are initialized (warm start / cold start)
	bInCopyCode : BOOL;  // if TRUE, the instance afterwards gets moved into the copy code (online change)
END_VAR
AddInput('in1',THIS^.in1);
AddInput('in2',THIS^.in2);
AddOutput('out', THIS^.out);
END_METHOD

METHOD PUBLIC Clone : I_Node
VAR
	pNode : POINTER TO ADD_LWORD;
END_VAR
pNode := __NEW(ADD_LWORD);
Clone := pNode^;
END_METHOD

METHOD PROTECTED OnExecute
VAR
END_VAR
out.Value := in1.Value + in2.Value;
END_METHOD

END_FUNCTION_BLOCK

// Core/Nodes/ADD/ADD_REAL
{attribute 'linkalways'} 
{attribute 'no_explicit_call' := 'This FB is a CLASS and must be accessed using methods or properties'}
{attribute 'enable_dynamic_creation'}
FUNCTION_BLOCK FINAL ADD_REAL EXTENDS Node
VAR
	in1 : _REAL(0.0);
	in2 : _REAL(0.0);
	out : _REAL(0.0);
END_VAR

METHOD FB_init : BOOL
VAR_INPUT
	bInitRetains : BOOL; // if TRUE, the retain variables are initialized (warm start / cold start)
	bInCopyCode : BOOL;  // if TRUE, the instance afterwards gets moved into the copy code (online change)
END_VAR
AddInput('in1',THIS^.in1);
AddInput('in2',THIS^.in2);
AddOutput('out', THIS^.out);
END_METHOD

METHOD PUBLIC Clone : I_Node
VAR
	pNode : POINTER TO ADD_REAL;
END_VAR
pNode := __NEW(ADD_REAL);
Clone := pNode^;
END_METHOD

METHOD PROTECTED OnExecute
VAR
END_VAR
out.Value := in1.Value + in2.Value;
END_METHOD

END_FUNCTION_BLOCK

// Core/Nodes/ADD/ADD_SINT
{attribute 'linkalways'} 
{attribute 'no_explicit_call' := 'This FB is a CLASS and must be accessed using methods or properties'}
{attribute 'enable_dynamic_creation'}
FUNCTION_BLOCK FINAL ADD_SINT EXTENDS Node
VAR
	in1 : _SINT(0);
	in2 : _SINT(0);
	out : _SINT(0);
END_VAR

METHOD FB_init : BOOL
VAR_INPUT
	bInitRetains : BOOL; // if TRUE, the retain variables are initialized (warm start / cold start)
	bInCopyCode : BOOL;  // if TRUE, the instance afterwards gets moved into the copy code (online change)
END_VAR
AddInput('in1',THIS^.in1);
AddInput('in2',THIS^.in2);
AddOutput('out', THIS^.out);
END_METHOD

METHOD PUBLIC Clone : I_Node
VAR
	pNode : POINTER TO ADD_SINT;
END_VAR
pNode := __NEW(ADD_SINT);
Clone := pNode^;
END_METHOD

METHOD PROTECTED OnExecute
VAR
END_VAR
out.Value := in1.Value + in2.Value;
END_METHOD

END_FUNCTION_BLOCK

// Core/Nodes/ADD/ADD_UDINT
{attribute 'linkalways'} 
{attribute 'no_explicit_call' := 'This FB is a CLASS and must be accessed using methods or properties'}
{attribute 'enable_dynamic_creation'}
FUNCTION_BLOCK FINAL ADD_UDINT EXTENDS Node
VAR
	in1 : _UDINT(0);
	in2 : _UDINT(0);
	out : _UDINT(0);
END_VAR

METHOD FB_init : BOOL
VAR_INPUT
	bInitRetains : BOOL; // if TRUE, the retain variables are initialized (warm start / cold start)
	bInCopyCode : BOOL;  // if TRUE, the instance afterwards gets moved into the copy code (online change)
END_VAR
AddInput('in1',THIS^.in1);
AddInput('in2',THIS^.in2);
AddOutput('out', THIS^.out);
END_METHOD

METHOD PUBLIC Clone : I_Node
VAR
	pNode : POINTER TO ADD_UDINT;
END_VAR
pNode := __NEW(ADD_UDINT);
Clone := pNode^;
END_METHOD

METHOD PROTECTED OnExecute
VAR
END_VAR
out.Value := in1.Value + in2.Value;
END_METHOD

END_FUNCTION_BLOCK

// Core/Nodes/ADD/ADD_UINT
{attribute 'linkalways'} 
{attribute 'no_explicit_call' := 'This FB is a CLASS and must be accessed using methods or properties'}
{attribute 'enable_dynamic_creation'}
FUNCTION_BLOCK FINAL ADD_UINT EXTENDS Node
VAR
	in1 : _UINT(0);
	in2 : _UINT(0);
	out : _UINT(0);
END_VAR

METHOD FB_init : BOOL
VAR_INPUT
	bInitRetains : BOOL; // if TRUE, the retain variables are initialized (warm start / cold start)
	bInCopyCode : BOOL;  // if TRUE, the instance afterwards gets moved into the copy code (online change)
END_VAR
AddInput('in1',THIS^.in1);
AddInput('in2',THIS^.in2);
AddOutput('out', THIS^.out);
END_METHOD

METHOD PUBLIC Clone : I_Node
VAR
	pNode : POINTER TO ADD_UINT;
END_VAR
pNode := __NEW(ADD_UINT);
Clone := pNode^;
END_METHOD

METHOD PROTECTED OnExecute
VAR
END_VAR
out.Value := in1.Value + in2.Value;
END_METHOD

END_FUNCTION_BLOCK

// Core/Nodes/ADD/ADD_ULINT
{attribute 'linkalways'} 
{attribute 'no_explicit_call' := 'This FB is a CLASS and must be accessed using methods or properties'}
{attribute 'enable_dynamic_creation'}
FUNCTION_BLOCK FINAL ADD_ULINT EXTENDS Node
VAR
	in1 : _ULINT(0);
	in2 : _ULINT(0);
	out : _ULINT(0);
END_VAR

METHOD FB_init : BOOL
VAR_INPUT
	bInitRetains : BOOL; // if TRUE, the retain variables are initialized (warm start / cold start)
	bInCopyCode : BOOL;  // if TRUE, the instance afterwards gets moved into the copy code (online change)
END_VAR
AddInput('in1',THIS^.in1);
AddInput('in2',THIS^.in2);
AddOutput('out', THIS^.out);
END_METHOD

METHOD PUBLIC Clone : I_Node
VAR
	pNode : POINTER TO ADD_ULINT;
END_VAR
pNode := __NEW(ADD_ULINT);
Clone := pNode^;
END_METHOD

METHOD PROTECTED OnExecute
VAR
END_VAR
out.Value := in1.Value + in2.Value;
END_METHOD

END_FUNCTION_BLOCK

// Core/Nodes/ADD/ADD_USINT
{attribute 'linkalways'} 
{attribute 'no_explicit_call' := 'This FB is a CLASS and must be accessed using methods or properties'}
{attribute 'enable_dynamic_creation'}
FUNCTION_BLOCK FINAL ADD_USINT EXTENDS Node
VAR
	in1 : _USINT(0);
	in2 : _USINT(0);
	out : _USINT(0);
END_VAR

METHOD FB_init : BOOL
VAR_INPUT
	bInitRetains : BOOL; // if TRUE, the retain variables are initialized (warm start / cold start)
	bInCopyCode : BOOL;  // if TRUE, the instance afterwards gets moved into the copy code (online change)
END_VAR
AddInput('in1',THIS^.in1);
AddInput('in2',THIS^.in2);
AddOutput('out', THIS^.out);
END_METHOD

METHOD PUBLIC Clone : I_Node
VAR
	pNode : POINTER TO ADD_USINT;
END_VAR
pNode := __NEW(ADD_USINT);
Clone := pNode^;
END_METHOD

METHOD PROTECTED OnExecute
VAR
END_VAR
out.Value := in1.Value + in2.Value;
END_METHOD

END_FUNCTION_BLOCK

// Core/Nodes/ADD/ADD_WORD
{attribute 'linkalways'} 
{attribute 'no_explicit_call' := 'This FB is a CLASS and must be accessed using methods or properties'}
{attribute 'enable_dynamic_creation'}
FUNCTION_BLOCK FINAL ADD_WORD EXTENDS Node
VAR
	in1 : _WORD(0);
	in2 : _WORD(0);
	out : _WORD(0);
END_VAR

METHOD FB_init : BOOL
VAR_INPUT
	bInitRetains : BOOL; // if TRUE, the retain variables are initialized (warm start / cold start)
	bInCopyCode : BOOL;  // if TRUE, the instance afterwards gets moved into the copy code (online change)
END_VAR
AddInput('in1',THIS^.in1);
AddInput('in2',THIS^.in2);
AddOutput('out', THIS^.out);
END_METHOD

METHOD PUBLIC Clone : I_Node
VAR
	pNode : POINTER TO ADD_WORD;
END_VAR
pNode := __NEW(ADD_WORD);
Clone := pNode^;
END_METHOD

METHOD PROTECTED OnExecute
VAR
END_VAR
out.Value := in1.Value + in2.Value;
END_METHOD

END_FUNCTION_BLOCK

// Core/Nodes/DIV/DIV_BYTE
{attribute 'linkalways'} 
{attribute 'no_explicit_call' := 'This FB is a CLASS and must be accessed using methods or properties'}
{attribute 'enable_dynamic_creation'}
FUNCTION_BLOCK FINAL DIV_BYTE EXTENDS Node
VAR
	in1 : _BYTE(0);
	in2 : _BYTE(0);
	out : _BYTE(0);
	div0 : _BOOL(FALSE);
END_VAR

METHOD FB_init : BOOL
VAR_INPUT
	bInitRetains : BOOL; // if TRUE, the retain variables are initialized (warm start / cold start)
	bInCopyCode : BOOL;  // if TRUE, the instance afterwards gets moved into the copy code (online change)
END_VAR
AddInput('in1',THIS^.in1);
AddInput('in2',THIS^.in2);
AddOutput('out', THIS^.out);
AddOutput('div0', THIS^.div0);
END_METHOD

METHOD PUBLIC Clone : I_Node
VAR
	pNode : POINTER TO DIV_BYTE;
END_VAR
pNode := __NEW(DIV_BYTE);
Clone := pNode^;
END_METHOD

METHOD PROTECTED OnExecute
VAR
END_VAR
IF in2.Value = 0 THEN
	div0.Value := TRUE;
	RETURN;
END_IF

out.Value := in1.Value / in2.Value;
div0.Value := FALSE;
END_METHOD

END_FUNCTION_BLOCK

// Core/Nodes/DIV/DIV_DINT
{attribute 'linkalways'} 
{attribute 'no_explicit_call' := 'This FB is a CLASS and must be accessed using methods or properties'}
{attribute 'enable_dynamic_creation'}
FUNCTION_BLOCK FINAL DIV_DINT EXTENDS Node
VAR
	in1 : _DINT(0);
	in2 : _DINT(0);
	out : _DINT(0);
	div0 : _BOOL(FALSE);
END_VAR

METHOD FB_init : BOOL
VAR_INPUT
	bInitRetains : BOOL; // if TRUE, the retain variables are initialized (warm start / cold start)
	bInCopyCode : BOOL;  // if TRUE, the instance afterwards gets moved into the copy code (online change)
END_VAR
AddInput('in1',THIS^.in1);
AddInput('in2',THIS^.in2);
AddOutput('out', THIS^.out);
AddOutput('div0', THIS^.div0);
END_METHOD

METHOD PUBLIC Clone : I_Node
VAR
	pNode : POINTER TO DIV_DINT;
END_VAR
pNode := __NEW(DIV_DINT);
Clone := pNode^;
END_METHOD

METHOD PROTECTED OnExecute
VAR
END_VAR
IF in2.Value = 0 THEN
	div0.Value := TRUE;
	RETURN;
END_IF

out.Value := in1.Value / in2.Value;
div0.Value := FALSE;
END_METHOD

END_FUNCTION_BLOCK

// Core/Nodes/DIV/DIV_DWORD
{attribute 'linkalways'} 
{attribute 'no_explicit_call' := 'This FB is a CLASS and must be accessed using methods or properties'}
{attribute 'enable_dynamic_creation'}
FUNCTION_BLOCK FINAL DIV_DWORD EXTENDS Node
VAR
	in1 : _DWORD(0);
	in2 : _DWORD(0);
	out : _DWORD(0);
	div0 : _BOOL(FALSE);
END_VAR

METHOD FB_init : BOOL
VAR_INPUT
	bInitRetains : BOOL; // if TRUE, the retain variables are initialized (warm start / cold start)
	bInCopyCode : BOOL;  // if TRUE, the instance afterwards gets moved into the copy code (online change)
END_VAR
AddInput('in1',THIS^.in1);
AddInput('in2',THIS^.in2);
AddOutput('out', THIS^.out);
AddOutput('div0', THIS^.div0);
END_METHOD

METHOD PUBLIC Clone : I_Node
VAR
	pNode : POINTER TO DIV_DWORD;
END_VAR
pNode := __NEW(DIV_DWORD);
Clone := pNode^;
END_METHOD

METHOD PROTECTED OnExecute
VAR
END_VAR
IF in2.Value = 0 THEN
	div0.Value := TRUE;
	RETURN;
END_IF

out.Value := in1.Value / in2.Value;
div0.Value := FALSE;
END_METHOD

END_FUNCTION_BLOCK

// Core/Nodes/DIV/DIV_INT
{attribute 'linkalways'} 
{attribute 'no_explicit_call' := 'This FB is a CLASS and must be accessed using methods or properties'}
{attribute 'enable_dynamic_creation'}
FUNCTION_BLOCK FINAL DIV_INT EXTENDS Node
VAR
	in1 : _INT(0);
	in2 : _INT(0);
	out : _INT(0);
	div0 : _BOOL(FALSE);
END_VAR

METHOD FB_init : BOOL
VAR_INPUT
	bInitRetains : BOOL; // if TRUE, the retain variables are initialized (warm start / cold start)
	bInCopyCode : BOOL;  // if TRUE, the instance afterwards gets moved into the copy code (online change)
END_VAR
AddInput('in1',THIS^.in1);
AddInput('in2',THIS^.in2);
AddOutput('out', THIS^.out);
AddOutput('div0', THIS^.div0);
END_METHOD

METHOD PUBLIC Clone : I_Node
VAR
	pNode : POINTER TO DIV_INT;
END_VAR
pNode := __NEW(DIV_INT);
Clone := pNode^;
END_METHOD

METHOD PROTECTED OnExecute
VAR
END_VAR
IF in2.Value = 0 THEN
	div0.Value := TRUE;
	RETURN;
END_IF

out.Value := in1.Value / in2.Value;
div0.Value := FALSE;
END_METHOD

END_FUNCTION_BLOCK

// Core/Nodes/DIV/DIV_LINT
{attribute 'linkalways'} 
{attribute 'no_explicit_call' := 'This FB is a CLASS and must be accessed using methods or properties'}
{attribute 'enable_dynamic_creation'}
FUNCTION_BLOCK FINAL DIV_LINT EXTENDS Node
VAR
	in1 : _LINT(0);
	in2 : _LINT(0);
	out : _LINT(0);
	div0 : _BOOL(FALSE);
END_VAR

METHOD FB_init : BOOL
VAR_INPUT
	bInitRetains : BOOL; // if TRUE, the retain variables are initialized (warm start / cold start)
	bInCopyCode : BOOL;  // if TRUE, the instance afterwards gets moved into the copy code (online change)
END_VAR
AddInput('in1',THIS^.in1);
AddInput('in2',THIS^.in2);
AddOutput('out', THIS^.out);
AddOutput('div0', THIS^.div0);
END_METHOD

METHOD PUBLIC Clone : I_Node
VAR
	pNode : POINTER TO DIV_LINT;
END_VAR
pNode := __NEW(DIV_LINT);
Clone := pNode^;
END_METHOD

METHOD PROTECTED OnExecute
VAR
END_VAR
IF in2.Value = 0 THEN
	div0.Value := TRUE;
	RETURN;
END_IF

out.Value := in1.Value / in2.Value;
div0.Value := FALSE;
END_METHOD

END_FUNCTION_BLOCK

// Core/Nodes/DIV/DIV_LREAL
{attribute 'linkalways'} 
{attribute 'no_explicit_call' := 'This FB is a CLASS and must be accessed using methods or properties'}
{attribute 'enable_dynamic_creation'}
FUNCTION_BLOCK FINAL DIV_LREAL EXTENDS Node
VAR
	in1 : _LREAL(0.0);
	in2 : _LREAL(0.0);
	out : _LREAL(0.0);
	div0 : _BOOL(FALSE);
END_VAR

METHOD FB_init : BOOL
VAR_INPUT
	bInitRetains : BOOL; // if TRUE, the retain variables are initialized (warm start / cold start)
	bInCopyCode : BOOL;  // if TRUE, the instance afterwards gets moved into the copy code (online change)
END_VAR
AddInput('in1',THIS^.in1);
AddInput('in2',THIS^.in2);
AddOutput('out', THIS^.out);
AddOutput('div0', THIS^.div0);
END_METHOD

METHOD PUBLIC Clone : I_Node
VAR
	pNode : POINTER TO DIV_LREAL;
END_VAR
pNode := __NEW(DIV_LREAL);
Clone := pNode^;
END_METHOD

METHOD PROTECTED OnExecute
VAR
END_VAR
IF in2.Value = 0 THEN
	div0.Value := TRUE;
	RETURN;
END_IF

out.Value := in1.Value / in2.Value;
div0.Value := FALSE;
END_METHOD

END_FUNCTION_BLOCK

// Core/Nodes/DIV/DIV_LWORD
{attribute 'linkalways'} 
{attribute 'no_explicit_call' := 'This FB is a CLASS and must be accessed using methods or properties'}
{attribute 'enable_dynamic_creation'}
FUNCTION_BLOCK FINAL DIV_LWORD EXTENDS Node
VAR
	in1 : _LWORD(0);
	in2 : _LWORD(0);
	out : _LWORD(0);
	div0 : _BOOL(FALSE);
END_VAR

METHOD FB_init : BOOL
VAR_INPUT
	bInitRetains : BOOL; // if TRUE, the retain variables are initialized (warm start / cold start)
	bInCopyCode : BOOL;  // if TRUE, the instance afterwards gets moved into the copy code (online change)
END_VAR
AddInput('in1',THIS^.in1);
AddInput('in2',THIS^.in2);
AddOutput('out', THIS^.out);
AddOutput('div0', THIS^.div0);
END_METHOD

METHOD PUBLIC Clone : I_Node
VAR
	pNode : POINTER TO DIV_LWORD;
END_VAR
pNode := __NEW(DIV_LWORD);
Clone := pNode^;
END_METHOD

METHOD PROTECTED OnExecute
VAR
END_VAR
IF in2.Value = 0 THEN
	div0.Value := TRUE;
	RETURN;
END_IF

out.Value := in1.Value / in2.Value;
div0.Value := FALSE;
END_METHOD

END_FUNCTION_BLOCK

// Core/Nodes/DIV/DIV_REAL
{attribute 'linkalways'} 
{attribute 'no_explicit_call' := 'This FB is a CLASS and must be accessed using methods or properties'}
{attribute 'enable_dynamic_creation'}
FUNCTION_BLOCK FINAL DIV_REAL EXTENDS Node
VAR
	in1 : _REAL(0.0);
	in2 : _REAL(0.0);
	out : _REAL(0.0);
	div0 : _BOOL(FALSE);
END_VAR

METHOD FB_init : BOOL
VAR_INPUT
	bInitRetains : BOOL; // if TRUE, the retain variables are initialized (warm start / cold start)
	bInCopyCode : BOOL;  // if TRUE, the instance afterwards gets moved into the copy code (online change)
END_VAR
AddInput('in1',THIS^.in1);
AddInput('in2',THIS^.in2);
AddOutput('out', THIS^.out);
AddOutput('div0', THIS^.div0);
END_METHOD

METHOD PUBLIC Clone : I_Node
VAR
	pNode : POINTER TO DIV_REAL;
END_VAR
pNode := __NEW(DIV_REAL);
Clone := pNode^;
END_METHOD

METHOD PROTECTED OnExecute
VAR
END_VAR
IF in2.Value = 0 THEN
	div0.Value := TRUE;
	RETURN;
END_IF

out.Value := in1.Value / in2.Value;
div0.Value := FALSE;
END_METHOD

END_FUNCTION_BLOCK

// Core/Nodes/DIV/DIV_SINT
{attribute 'linkalways'} 
{attribute 'no_explicit_call' := 'This FB is a CLASS and must be accessed using methods or properties'}
{attribute 'enable_dynamic_creation'}
FUNCTION_BLOCK FINAL DIV_SINT EXTENDS Node
VAR
	in1 : _SINT(0);
	in2 : _SINT(0);
	out : _SINT(0);
	div0 : _BOOL(FALSE);
END_VAR

METHOD FB_init : BOOL
VAR_INPUT
	bInitRetains : BOOL; // if TRUE, the retain variables are initialized (warm start / cold start)
	bInCopyCode : BOOL;  // if TRUE, the instance afterwards gets moved into the copy code (online change)
END_VAR
AddInput('in1',THIS^.in1);
AddInput('in2',THIS^.in2);
AddOutput('out', THIS^.out);
AddOutput('div0', THIS^.div0);
END_METHOD

METHOD PUBLIC Clone : I_Node
VAR
	pNode : POINTER TO DIV_SINT;
END_VAR
pNode := __NEW(DIV_SINT);
Clone := pNode^;
END_METHOD

METHOD PROTECTED OnExecute
VAR
END_VAR
IF in2.Value = 0 THEN
	div0.Value := TRUE;
	RETURN;
END_IF

out.Value := in1.Value / in2.Value;
div0.Value := FALSE;
END_METHOD

END_FUNCTION_BLOCK

// Core/Nodes/DIV/DIV_UDINT
{attribute 'linkalways'} 
{attribute 'no_explicit_call' := 'This FB is a CLASS and must be accessed using methods or properties'}
{attribute 'enable_dynamic_creation'}
FUNCTION_BLOCK FINAL DIV_UDINT EXTENDS Node
VAR
	in1 : _UDINT(0);
	in2 : _UDINT(0);
	out : _UDINT(0);
	div0 : _BOOL(FALSE);
END_VAR

METHOD FB_init : BOOL
VAR_INPUT
	bInitRetains : BOOL; // if TRUE, the retain variables are initialized (warm start / cold start)
	bInCopyCode : BOOL;  // if TRUE, the instance afterwards gets moved into the copy code (online change)
END_VAR
AddInput('in1',THIS^.in1);
AddInput('in2',THIS^.in2);
AddOutput('out', THIS^.out);
AddOutput('div0', THIS^.div0);
END_METHOD

METHOD PUBLIC Clone : I_Node
VAR
	pNode : POINTER TO DIV_UDINT;
END_VAR
pNode := __NEW(DIV_UDINT);
Clone := pNode^;
END_METHOD

METHOD PROTECTED OnExecute
VAR
END_VAR
IF in2.Value = 0 THEN
	div0.Value := TRUE;
	RETURN;
END_IF

out.Value := in1.Value / in2.Value;
div0.Value := FALSE;
END_METHOD

END_FUNCTION_BLOCK

// Core/Nodes/DIV/DIV_UINT
{attribute 'linkalways'} 
{attribute 'no_explicit_call' := 'This FB is a CLASS and must be accessed using methods or properties'}
{attribute 'enable_dynamic_creation'}
FUNCTION_BLOCK FINAL DIV_UINT EXTENDS Node
VAR
	in1 : _UINT(0);
	in2 : _UINT(0);
	out : _UINT(0);
	div0 : _BOOL(FALSE);
END_VAR

METHOD FB_init : BOOL
VAR_INPUT
	bInitRetains : BOOL; // if TRUE, the retain variables are initialized (warm start / cold start)
	bInCopyCode : BOOL;  // if TRUE, the instance afterwards gets moved into the copy code (online change)
END_VAR
AddInput('in1',THIS^.in1);
AddInput('in2',THIS^.in2);
AddOutput('out', THIS^.out);
AddOutput('div0', THIS^.div0);
END_METHOD

METHOD PUBLIC Clone : I_Node
VAR
	pNode : POINTER TO DIV_UINT;
END_VAR
pNode := __NEW(DIV_UINT);
Clone := pNode^;
END_METHOD

METHOD PROTECTED OnExecute
VAR
END_VAR
IF in2.Value = 0 THEN
	div0.Value := TRUE;
	RETURN;
END_IF

out.Value := in1.Value / in2.Value;
div0.Value := FALSE;
END_METHOD

END_FUNCTION_BLOCK

// Core/Nodes/DIV/DIV_ULINT
{attribute 'linkalways'} 
{attribute 'no_explicit_call' := 'This FB is a CLASS and must be accessed using methods or properties'}
{attribute 'enable_dynamic_creation'}
FUNCTION_BLOCK FINAL DIV_ULINT EXTENDS Node
VAR
	in1 : _ULINT(0);
	in2 : _ULINT(0);
	out : _ULINT(0);
	div0 : _BOOL(FALSE);
END_VAR

METHOD FB_init : BOOL
VAR_INPUT
	bInitRetains : BOOL; // if TRUE, the retain variables are initialized (warm start / cold start)
	bInCopyCode : BOOL;  // if TRUE, the instance afterwards gets moved into the copy code (online change)
END_VAR
AddInput('in1',THIS^.in1);
AddInput('in2',THIS^.in2);
AddOutput('out', THIS^.out);
AddOutput('div0', THIS^.div0);
END_METHOD

METHOD PUBLIC Clone : I_Node
VAR
	pNode : POINTER TO DIV_ULINT;
END_VAR
pNode := __NEW(DIV_ULINT);
Clone := pNode^;
END_METHOD

METHOD PROTECTED OnExecute
VAR
END_VAR
IF in2.Value = 0 THEN
	div0.Value := TRUE;
	RETURN;
END_IF

out.Value := in1.Value / in2.Value;
div0.Value := FALSE;
END_METHOD

END_FUNCTION_BLOCK

// Core/Nodes/DIV/DIV_USINT
{attribute 'linkalways'} 
{attribute 'no_explicit_call' := 'This FB is a CLASS and must be accessed using methods or properties'}
{attribute 'enable_dynamic_creation'}
FUNCTION_BLOCK FINAL DIV_USINT EXTENDS Node
VAR
	in1 : _USINT(0);
	in2 : _USINT(0);
	out : _USINT(0);
	div0 : _BOOL(FALSE);
END_VAR

METHOD FB_init : BOOL
VAR_INPUT
	bInitRetains : BOOL; // if TRUE, the retain variables are initialized (warm start / cold start)
	bInCopyCode : BOOL;  // if TRUE, the instance afterwards gets moved into the copy code (online change)
END_VAR
AddInput('in1',THIS^.in1);
AddInput('in2',THIS^.in2);
AddOutput('out', THIS^.out);
AddOutput('div0', THIS^.div0);
END_METHOD

METHOD PUBLIC Clone : I_Node
VAR
	pNode : POINTER TO DIV_USINT;
END_VAR
pNode := __NEW(DIV_USINT);
Clone := pNode^;
END_METHOD

METHOD PROTECTED OnExecute
VAR
END_VAR
IF in2.Value = 0 THEN
	div0.Value := TRUE;
	RETURN;
END_IF

out.Value := in1.Value / in2.Value;
div0.Value := FALSE;
END_METHOD

END_FUNCTION_BLOCK

// Core/Nodes/DIV/DIV_WORD
{attribute 'linkalways'} 
{attribute 'no_explicit_call' := 'This FB is a CLASS and must be accessed using methods or properties'}
{attribute 'enable_dynamic_creation'}
FUNCTION_BLOCK FINAL DIV_WORD EXTENDS Node
VAR
	in1 : _WORD(0);
	in2 : _WORD(0);
	out : _WORD(0);
	div0 : _BOOL(FALSE);
END_VAR

METHOD FB_init : BOOL
VAR_INPUT
	bInitRetains : BOOL; // if TRUE, the retain variables are initialized (warm start / cold start)
	bInCopyCode : BOOL;  // if TRUE, the instance afterwards gets moved into the copy code (online change)
END_VAR
AddInput('in1',THIS^.in1);
AddInput('in2',THIS^.in2);
AddOutput('out', THIS^.out);
AddOutput('div0', THIS^.div0);
END_METHOD

METHOD PUBLIC Clone : I_Node
VAR
	pNode : POINTER TO DIV_WORD;
END_VAR
pNode := __NEW(DIV_WORD);
Clone := pNode^;
END_METHOD

METHOD PROTECTED OnExecute
VAR
END_VAR
IF in2.Value = 0 THEN
	div0.Value := TRUE;
	RETURN;
END_IF

out.Value := in1.Value / in2.Value;
div0.Value := FALSE;
END_METHOD

END_FUNCTION_BLOCK

// Core/Nodes/MOD/MOD_BYTE
{attribute 'linkalways'} 
{attribute 'no_explicit_call' := 'This FB is a CLASS and must be accessed using methods or properties'}
{attribute 'enable_dynamic_creation'}
FUNCTION_BLOCK FINAL MOD_BYTE EXTENDS Node
VAR
	in1 : _BYTE(0);
	in2 : _BYTE(0);
	out : _BYTE(0);
END_VAR

METHOD FB_init : BOOL
VAR_INPUT
	bInitRetains : BOOL; // if TRUE, the retain variables are initialized (warm start / cold start)
	bInCopyCode : BOOL;  // if TRUE, the instance afterwards gets moved into the copy code (online change)
END_VAR
AddInput('in1',THIS^.in1);
AddInput('in2',THIS^.in2);
AddOutput('out', THIS^.out);
END_METHOD

METHOD PUBLIC Clone : I_Node
VAR
	pNode : POINTER TO MOD_BYTE;
END_VAR
pNode := __NEW(MOD_BYTE);
Clone := pNode^;
END_METHOD

METHOD PROTECTED OnExecute
VAR
END_VAR
out.Value := in1.Value MOD in2.Value;
END_METHOD

END_FUNCTION_BLOCK

// Core/Nodes/MOD/MOD_DINT
{attribute 'linkalways'} 
{attribute 'no_explicit_call' := 'This FB is a CLASS and must be accessed using methods or properties'}
{attribute 'enable_dynamic_creation'}
FUNCTION_BLOCK FINAL MOD_DINT EXTENDS Node
VAR
	in1 : _DINT(0);
	in2 : _DINT(0);
	out : _DINT(0);
END_VAR

METHOD FB_init : BOOL
VAR_INPUT
	bInitRetains : BOOL; // if TRUE, the retain variables are initialized (warm start / cold start)
	bInCopyCode : BOOL;  // if TRUE, the instance afterwards gets moved into the copy code (online change)
END_VAR
AddInput('in1',THIS^.in1);
AddInput('in2',THIS^.in2);
AddOutput('out', THIS^.out);
END_METHOD

METHOD PUBLIC Clone : I_Node
VAR
	pNode : POINTER TO MOD_DINT;
END_VAR
pNode := __NEW(MOD_DINT);
Clone := pNode^;
END_METHOD

METHOD PROTECTED OnExecute
VAR
END_VAR
out.Value := in1.Value MOD in2.Value;
END_METHOD

END_FUNCTION_BLOCK

// Core/Nodes/MOD/MOD_DWORD
{attribute 'linkalways'} 
{attribute 'no_explicit_call' := 'This FB is a CLASS and must be accessed using methods or properties'}
{attribute 'enable_dynamic_creation'}
FUNCTION_BLOCK FINAL MOD_DWORD EXTENDS Node
VAR
	in1 : _DWORD(0);
	in2 : _DWORD(0);
	out : _DWORD(0);
END_VAR

METHOD FB_init : BOOL
VAR_INPUT
	bInitRetains : BOOL; // if TRUE, the retain variables are initialized (warm start / cold start)
	bInCopyCode : BOOL;  // if TRUE, the instance afterwards gets moved into the copy code (online change)
END_VAR
AddInput('in1',THIS^.in1);
AddInput('in2',THIS^.in2);
AddOutput('out', THIS^.out);
END_METHOD

METHOD PUBLIC Clone : I_Node
VAR
	pNode : POINTER TO MOD_DWORD;
END_VAR
pNode := __NEW(MOD_DWORD);
Clone := pNode^;
END_METHOD

METHOD PROTECTED OnExecute
VAR
END_VAR
out.Value := in1.Value MOD in2.Value;
END_METHOD

END_FUNCTION_BLOCK

// Core/Nodes/MOD/MOD_INT
{attribute 'linkalways'} 
{attribute 'no_explicit_call' := 'This FB is a CLASS and must be accessed using methods or properties'}
{attribute 'enable_dynamic_creation'}
FUNCTION_BLOCK FINAL MOD_INT EXTENDS Node
VAR
	in1 : _INT(0);
	in2 : _INT(0);
	out : _INT(0);
END_VAR

METHOD FB_init : BOOL
VAR_INPUT
	bInitRetains : BOOL; // if TRUE, the retain variables are initialized (warm start / cold start)
	bInCopyCode : BOOL;  // if TRUE, the instance afterwards gets moved into the copy code (online change)
END_VAR
AddInput('in1',THIS^.in1);
AddInput('in2',THIS^.in2);
AddOutput('out', THIS^.out);
END_METHOD

METHOD PUBLIC Clone : I_Node
VAR
	pNode : POINTER TO MOD_INT;
END_VAR
pNode := __NEW(MOD_INT);
Clone := pNode^;
END_METHOD

METHOD PROTECTED OnExecute
VAR
END_VAR
out.Value := in1.Value MOD in2.Value;
END_METHOD

END_FUNCTION_BLOCK

// Core/Nodes/MOD/MOD_LINT
{attribute 'linkalways'} 
{attribute 'no_explicit_call' := 'This FB is a CLASS and must be accessed using methods or properties'}
{attribute 'enable_dynamic_creation'}
FUNCTION_BLOCK FINAL MOD_LINT EXTENDS Node
VAR
	in1 : _LINT(0);
	in2 : _LINT(0);
	out : _LINT(0);
END_VAR

METHOD FB_init : BOOL
VAR_INPUT
	bInitRetains : BOOL; // if TRUE, the retain variables are initialized (warm start / cold start)
	bInCopyCode : BOOL;  // if TRUE, the instance afterwards gets moved into the copy code (online change)
END_VAR
AddInput('in1',THIS^.in1);
AddInput('in2',THIS^.in2);
AddOutput('out', THIS^.out);
END_METHOD

METHOD PUBLIC Clone : I_Node
VAR
	pNode : POINTER TO MOD_LINT;
END_VAR
pNode := __NEW(MOD_LINT);
Clone := pNode^;
END_METHOD

METHOD PROTECTED OnExecute
VAR
END_VAR
out.Value := in1.Value MOD in2.Value;
END_METHOD

END_FUNCTION_BLOCK

// Core/Nodes/MOD/MOD_LREAL
{attribute 'linkalways'} 
{attribute 'no_explicit_call' := 'This FB is a CLASS and must be accessed using methods or properties'}
{attribute 'enable_dynamic_creation'}
FUNCTION_BLOCK FINAL MOD_LREAL EXTENDS Node
VAR
	in1 : _LREAL(0.0);
	in2 : _LREAL(0.0);
	out : _LREAL(0.0);
END_VAR

METHOD FB_init : BOOL
VAR_INPUT
	bInitRetains : BOOL; // if TRUE, the retain variables are initialized (warm start / cold start)
	bInCopyCode : BOOL;  // if TRUE, the instance afterwards gets moved into the copy code (online change)
END_VAR
AddInput('in1',THIS^.in1);
AddInput('in2',THIS^.in2);
AddOutput('out', THIS^.out);
END_METHOD

METHOD PUBLIC Clone : I_Node
VAR
	pNode : POINTER TO MOD_LREAL;
END_VAR
pNode := __NEW(MOD_LREAL);
Clone := pNode^;
END_METHOD

METHOD PROTECTED OnExecute
VAR
END_VAR
out.Value := LMOD(in1.Value, in2.Value);
END_METHOD

END_FUNCTION_BLOCK

// Core/Nodes/MOD/MOD_LWORD
{attribute 'linkalways'} 
{attribute 'no_explicit_call' := 'This FB is a CLASS and must be accessed using methods or properties'}
{attribute 'enable_dynamic_creation'}
FUNCTION_BLOCK FINAL MOD_LWORD EXTENDS Node
VAR
	in1 : _LWORD(0);
	in2 : _LWORD(0);
	out : _LWORD(0);
END_VAR

METHOD FB_init : BOOL
VAR_INPUT
	bInitRetains : BOOL; // if TRUE, the retain variables are initialized (warm start / cold start)
	bInCopyCode : BOOL;  // if TRUE, the instance afterwards gets moved into the copy code (online change)
END_VAR
AddInput('in1',THIS^.in1);
AddInput('in2',THIS^.in2);
AddOutput('out', THIS^.out);
END_METHOD

METHOD PUBLIC Clone : I_Node
VAR
	pNode : POINTER TO MOD_LWORD;
END_VAR
pNode := __NEW(MOD_LWORD);
Clone := pNode^;
END_METHOD

METHOD PROTECTED OnExecute
VAR
END_VAR
out.Value := in1.Value MOD in2.Value;
END_METHOD

END_FUNCTION_BLOCK

// Core/Nodes/MOD/MOD_SINT
{attribute 'linkalways'} 
{attribute 'no_explicit_call' := 'This FB is a CLASS and must be accessed using methods or properties'}
{attribute 'enable_dynamic_creation'}
FUNCTION_BLOCK FINAL MOD_SINT EXTENDS Node
VAR
	in1 : _SINT(0);
	in2 : _SINT(0);
	out : _SINT(0);
END_VAR

METHOD FB_init : BOOL
VAR_INPUT
	bInitRetains : BOOL; // if TRUE, the retain variables are initialized (warm start / cold start)
	bInCopyCode : BOOL;  // if TRUE, the instance afterwards gets moved into the copy code (online change)
END_VAR
AddInput('in1',THIS^.in1);
AddInput('in2',THIS^.in2);
AddOutput('out', THIS^.out);
END_METHOD

METHOD PUBLIC Clone : I_Node
VAR
	pNode : POINTER TO MOD_SINT;
END_VAR
pNode := __NEW(MOD_SINT);
Clone := pNode^;
END_METHOD

METHOD PROTECTED OnExecute
VAR
END_VAR
out.Value := in1.Value MOD in2.Value;
END_METHOD

END_FUNCTION_BLOCK

// Core/Nodes/MOD/MOD_UDINT
{attribute 'linkalways'} 
{attribute 'no_explicit_call' := 'This FB is a CLASS and must be accessed using methods or properties'}
{attribute 'enable_dynamic_creation'}
FUNCTION_BLOCK FINAL MOD_UDINT EXTENDS Node
VAR
	in1 : _UDINT(0);
	in2 : _UDINT(0);
	out : _UDINT(0);
END_VAR

METHOD FB_init : BOOL
VAR_INPUT
	bInitRetains : BOOL; // if TRUE, the retain variables are initialized (warm start / cold start)
	bInCopyCode : BOOL;  // if TRUE, the instance afterwards gets moved into the copy code (online change)
END_VAR
AddInput('in1',THIS^.in1);
AddInput('in2',THIS^.in2);
AddOutput('out', THIS^.out);
END_METHOD

METHOD PUBLIC Clone : I_Node
VAR
	pNode : POINTER TO MOD_UDINT;
END_VAR
pNode := __NEW(MOD_UDINT);
Clone := pNode^;
END_METHOD

METHOD PROTECTED OnExecute
VAR
END_VAR
out.Value := in1.Value MOD in2.Value;
END_METHOD

END_FUNCTION_BLOCK

// Core/Nodes/MOD/MOD_UINT
{attribute 'linkalways'} 
{attribute 'no_explicit_call' := 'This FB is a CLASS and must be accessed using methods or properties'}
{attribute 'enable_dynamic_creation'}
FUNCTION_BLOCK FINAL MOD_UINT EXTENDS Node
VAR
	in1 : _UINT(0);
	in2 : _UINT(0);
	out : _UINT(0);
END_VAR

METHOD FB_init : BOOL
VAR_INPUT
	bInitRetains : BOOL; // if TRUE, the retain variables are initialized (warm start / cold start)
	bInCopyCode : BOOL;  // if TRUE, the instance afterwards gets moved into the copy code (online change)
END_VAR
AddInput('in1',THIS^.in1);
AddInput('in2',THIS^.in2);
AddOutput('out', THIS^.out);
END_METHOD

METHOD PUBLIC Clone : I_Node
VAR
	pNode : POINTER TO MOD_UINT;
END_VAR
pNode := __NEW(MOD_UINT);
Clone := pNode^;
END_METHOD

METHOD PROTECTED OnExecute
VAR
END_VAR
out.Value := in1.Value MOD in2.Value;
END_METHOD

END_FUNCTION_BLOCK

// Core/Nodes/MOD/MOD_ULINT
{attribute 'linkalways'} 
{attribute 'no_explicit_call' := 'This FB is a CLASS and must be accessed using methods or properties'}
{attribute 'enable_dynamic_creation'}
FUNCTION_BLOCK FINAL MOD_ULINT EXTENDS Node
VAR
	in1 : _ULINT(0);
	in2 : _ULINT(0);
	out : _ULINT(0);
END_VAR

METHOD FB_init : BOOL
VAR_INPUT
	bInitRetains : BOOL; // if TRUE, the retain variables are initialized (warm start / cold start)
	bInCopyCode : BOOL;  // if TRUE, the instance afterwards gets moved into the copy code (online change)
END_VAR
AddInput('in1',THIS^.in1);
AddInput('in2',THIS^.in2);
AddOutput('out', THIS^.out);
END_METHOD

METHOD PUBLIC Clone : I_Node
VAR
	pNode : POINTER TO MOD_ULINT;
END_VAR
pNode := __NEW(MOD_ULINT);
Clone := pNode^;
END_METHOD

METHOD PROTECTED OnExecute
VAR
END_VAR
out.Value := in1.Value MOD in2.Value;
END_METHOD

END_FUNCTION_BLOCK

// Core/Nodes/MOD/MOD_USINT
{attribute 'linkalways'} 
{attribute 'no_explicit_call' := 'This FB is a CLASS and must be accessed using methods or properties'}
{attribute 'enable_dynamic_creation'}
FUNCTION_BLOCK FINAL MOD_USINT EXTENDS Node
VAR
	in1 : _USINT(0);
	in2 : _USINT(0);
	out : _USINT(0);
END_VAR

METHOD FB_init : BOOL
VAR_INPUT
	bInitRetains : BOOL; // if TRUE, the retain variables are initialized (warm start / cold start)
	bInCopyCode : BOOL;  // if TRUE, the instance afterwards gets moved into the copy code (online change)
END_VAR
AddInput('in1',THIS^.in1);
AddInput('in2',THIS^.in2);
AddOutput('out', THIS^.out);
END_METHOD

METHOD PUBLIC Clone : I_Node
VAR
	pNode : POINTER TO MOD_USINT;
END_VAR
pNode := __NEW(MOD_USINT);
Clone := pNode^;
END_METHOD

METHOD PROTECTED OnExecute
VAR
END_VAR
out.Value := in1.Value MOD in2.Value;
END_METHOD

END_FUNCTION_BLOCK

// Core/Nodes/MOD/MOD_WORD
{attribute 'linkalways'} 
{attribute 'no_explicit_call' := 'This FB is a CLASS and must be accessed using methods or properties'}
{attribute 'enable_dynamic_creation'}
FUNCTION_BLOCK FINAL MOD_WORD EXTENDS Node
VAR
	in1 : _WORD(0);
	in2 : _WORD(0);
	out : _WORD(0);
END_VAR

METHOD FB_init : BOOL
VAR_INPUT
	bInitRetains : BOOL; // if TRUE, the retain variables are initialized (warm start / cold start)
	bInCopyCode : BOOL;  // if TRUE, the instance afterwards gets moved into the copy code (online change)
END_VAR
AddInput('in1',THIS^.in1);
AddInput('in2',THIS^.in2);
AddOutput('out', THIS^.out);
END_METHOD

METHOD PUBLIC Clone : I_Node
VAR
	pNode : POINTER TO MOD_WORD;
END_VAR
pNode := __NEW(MOD_WORD);
Clone := pNode^;
END_METHOD

METHOD PROTECTED OnExecute
VAR
END_VAR
out.Value := in1.Value MOD in2.Value;
END_METHOD

END_FUNCTION_BLOCK

// Core/Nodes/MUL/MUL_BYTE
{attribute 'linkalways'} 
{attribute 'no_explicit_call' := 'This FB is a CLASS and must be accessed using methods or properties'}
{attribute 'enable_dynamic_creation'}
FUNCTION_BLOCK FINAL MUL_BYTE EXTENDS Node
VAR
	in1 : _BYTE(0);
	in2 : _BYTE(0);
	out : _BYTE(0);
END_VAR

METHOD FB_init : BOOL
VAR_INPUT
	bInitRetains : BOOL; // if TRUE, the retain variables are initialized (warm start / cold start)
	bInCopyCode : BOOL;  // if TRUE, the instance afterwards gets moved into the copy code (online change)
END_VAR
AddInput('in1',THIS^.in1);
AddInput('in2',THIS^.in2);
AddOutput('out', THIS^.out);
END_METHOD

METHOD PUBLIC Clone : I_Node
VAR
	pNode : POINTER TO MUL_BYTE;
END_VAR
pNode := __NEW(MUL_BYTE);
Clone := pNode^;
END_METHOD

METHOD PROTECTED OnExecute
VAR
END_VAR
out.Value := in1.Value * in2.Value;
END_METHOD

END_FUNCTION_BLOCK

// Core/Nodes/MUL/MUL_DINT
{attribute 'linkalways'} 
{attribute 'no_explicit_call' := 'This FB is a CLASS and must be accessed using methods or properties'}
{attribute 'enable_dynamic_creation'}
FUNCTION_BLOCK FINAL MUL_DINT EXTENDS Node
VAR
	in1 : _DINT(0);
	in2 : _DINT(0);
	out : _DINT(0);
END_VAR

METHOD FB_init : BOOL
VAR_INPUT
	bInitRetains : BOOL; // if TRUE, the retain variables are initialized (warm start / cold start)
	bInCopyCode : BOOL;  // if TRUE, the instance afterwards gets moved into the copy code (online change)
END_VAR
AddInput('in1',THIS^.in1);
AddInput('in2',THIS^.in2);
AddOutput('out', THIS^.out);
END_METHOD

METHOD PUBLIC Clone : I_Node
VAR
	pNode : POINTER TO MUL_DINT;
END_VAR
pNode := __NEW(MUL_DINT);
Clone := pNode^;
END_METHOD

METHOD PROTECTED OnExecute
VAR
END_VAR
out.Value := in1.Value * in2.Value;
END_METHOD

END_FUNCTION_BLOCK

// Core/Nodes/MUL/MUL_DWORD
{attribute 'linkalways'} 
{attribute 'no_explicit_call' := 'This FB is a CLASS and must be accessed using methods or properties'}
{attribute 'enable_dynamic_creation'}
FUNCTION_BLOCK FINAL MUL_DWORD EXTENDS Node
VAR
	in1 : _DWORD(0);
	in2 : _DWORD(0);
	out : _DWORD(0);
END_VAR

METHOD FB_init : BOOL
VAR_INPUT
	bInitRetains : BOOL; // if TRUE, the retain variables are initialized (warm start / cold start)
	bInCopyCode : BOOL;  // if TRUE, the instance afterwards gets moved into the copy code (online change)
END_VAR
AddInput('in1',THIS^.in1);
AddInput('in2',THIS^.in2);
AddOutput('out', THIS^.out);
END_METHOD

METHOD PUBLIC Clone : I_Node
VAR
	pNode : POINTER TO MUL_DWORD;
END_VAR
pNode := __NEW(MUL_DWORD);
Clone := pNode^;
END_METHOD

METHOD PROTECTED OnExecute
VAR
END_VAR
out.Value := in1.Value * in2.Value;
END_METHOD

END_FUNCTION_BLOCK

// Core/Nodes/MUL/MUL_INT
{attribute 'linkalways'} 
{attribute 'no_explicit_call' := 'This FB is a CLASS and must be accessed using methods or properties'}
{attribute 'enable_dynamic_creation'}
FUNCTION_BLOCK FINAL MUL_INT EXTENDS Node
VAR
	in1 : _INT(0);
	in2 : _INT(0);
	out : _INT(0);
END_VAR

METHOD FB_init : BOOL
VAR_INPUT
	bInitRetains : BOOL; // if TRUE, the retain variables are initialized (warm start / cold start)
	bInCopyCode : BOOL;  // if TRUE, the instance afterwards gets moved into the copy code (online change)
END_VAR
AddInput('in1',THIS^.in1);
AddInput('in2',THIS^.in2);
AddOutput('out', THIS^.out);
END_METHOD

METHOD PUBLIC Clone : I_Node
VAR
	pNode : POINTER TO MUL_INT;
END_VAR
pNode := __NEW(MUL_INT);
Clone := pNode^;
END_METHOD

METHOD PROTECTED OnExecute
VAR
END_VAR
out.Value := in1.Value * in2.Value;
END_METHOD

END_FUNCTION_BLOCK

// Core/Nodes/MUL/MUL_LINT
{attribute 'linkalways'} 
{attribute 'no_explicit_call' := 'This FB is a CLASS and must be accessed using methods or properties'}
{attribute 'enable_dynamic_creation'}
FUNCTION_BLOCK FINAL MUL_LINT EXTENDS Node
VAR
	in1 : _LINT(0);
	in2 : _LINT(0);
	out : _LINT(0);
END_VAR

METHOD FB_init : BOOL
VAR_INPUT
	bInitRetains : BOOL; // if TRUE, the retain variables are initialized (warm start / cold start)
	bInCopyCode : BOOL;  // if TRUE, the instance afterwards gets moved into the copy code (online change)
END_VAR
AddInput('in1',THIS^.in1);
AddInput('in2',THIS^.in2);
AddOutput('out', THIS^.out);
END_METHOD

METHOD PUBLIC Clone : I_Node
VAR
	pNode : POINTER TO MUL_LINT;
END_VAR
pNode := __NEW(MUL_LINT);
Clone := pNode^;
END_METHOD

METHOD PROTECTED OnExecute
VAR
END_VAR
out.Value := in1.Value * in2.Value;
END_METHOD

END_FUNCTION_BLOCK

// Core/Nodes/MUL/MUL_LREAL
{attribute 'linkalways'} 
{attribute 'no_explicit_call' := 'This FB is a CLASS and must be accessed using methods or properties'}
{attribute 'enable_dynamic_creation'}
FUNCTION_BLOCK FINAL MUL_LREAL EXTENDS Node
VAR
	in1 : _LREAL(0.0);
	in2 : _LREAL(0.0);
	out : _LREAL(0.0);
END_VAR

METHOD FB_init : BOOL
VAR_INPUT
	bInitRetains : BOOL; // if TRUE, the retain variables are initialized (warm start / cold start)
	bInCopyCode : BOOL;  // if TRUE, the instance afterwards gets moved into the copy code (online change)
END_VAR
AddInput('in1',THIS^.in1);
AddInput('in2',THIS^.in2);
AddOutput('out', THIS^.out);
END_METHOD

METHOD PUBLIC Clone : I_Node
VAR
	pNode : POINTER TO MUL_LREAL;
END_VAR
pNode := __NEW(MUL_LREAL);
Clone := pNode^;
END_METHOD

METHOD PROTECTED OnExecute
VAR
END_VAR
out.Value := in1.Value * in2.Value;
END_METHOD

END_FUNCTION_BLOCK

// Core/Nodes/MUL/MUL_LWORD
{attribute 'linkalways'} 
{attribute 'no_explicit_call' := 'This FB is a CLASS and must be accessed using methods or properties'}
{attribute 'enable_dynamic_creation'}
FUNCTION_BLOCK FINAL MUL_LWORD EXTENDS Node
VAR
	in1 : _LWORD(0);
	in2 : _LWORD(0);
	out : _LWORD(0);
END_VAR

METHOD FB_init : BOOL
VAR_INPUT
	bInitRetains : BOOL; // if TRUE, the retain variables are initialized (warm start / cold start)
	bInCopyCode : BOOL;  // if TRUE, the instance afterwards gets moved into the copy code (online change)
END_VAR
AddInput('in1',THIS^.in1);
AddInput('in2',THIS^.in2);
AddOutput('out', THIS^.out);
END_METHOD

METHOD PUBLIC Clone : I_Node
VAR
	pNode : POINTER TO MUL_LWORD;
END_VAR
pNode := __NEW(MUL_LWORD);
Clone := pNode^;
END_METHOD

METHOD PROTECTED OnExecute
VAR
END_VAR
out.Value := in1.Value * in2.Value;
END_METHOD

END_FUNCTION_BLOCK

// Core/Nodes/MUL/MUL_REAL
{attribute 'linkalways'} 
{attribute 'no_explicit_call' := 'This FB is a CLASS and must be accessed using methods or properties'}
{attribute 'enable_dynamic_creation'}
FUNCTION_BLOCK FINAL MUL_REAL EXTENDS Node
VAR
	in1 : _REAL(0.0);
	in2 : _REAL(0.0);
	out : _REAL(0.0);
END_VAR

METHOD FB_init : BOOL
VAR_INPUT
	bInitRetains : BOOL; // if TRUE, the retain variables are initialized (warm start / cold start)
	bInCopyCode : BOOL;  // if TRUE, the instance afterwards gets moved into the copy code (online change)
END_VAR
AddInput('in1',THIS^.in1);
AddInput('in2',THIS^.in2);
AddOutput('out', THIS^.out);
END_METHOD

METHOD PUBLIC Clone : I_Node
VAR
	pNode : POINTER TO MUL_REAL;
END_VAR
pNode := __NEW(MUL_REAL);
Clone := pNode^;
END_METHOD

METHOD PROTECTED OnExecute
VAR
END_VAR
out.Value := in1.Value * in2.Value;
END_METHOD

END_FUNCTION_BLOCK

// Core/Nodes/MUL/MUL_SINT
{attribute 'linkalways'} 
{attribute 'no_explicit_call' := 'This FB is a CLASS and must be accessed using methods or properties'}
{attribute 'enable_dynamic_creation'}
FUNCTION_BLOCK FINAL MUL_SINT EXTENDS Node
VAR
	in1 : _SINT(0);
	in2 : _SINT(0);
	out : _SINT(0);
END_VAR

METHOD FB_init : BOOL
VAR_INPUT
	bInitRetains : BOOL; // if TRUE, the retain variables are initialized (warm start / cold start)
	bInCopyCode : BOOL;  // if TRUE, the instance afterwards gets moved into the copy code (online change)
END_VAR
AddInput('in1',THIS^.in1);
AddInput('in2',THIS^.in2);
AddOutput('out', THIS^.out);
END_METHOD

METHOD PUBLIC Clone : I_Node
VAR
	pNode : POINTER TO MUL_SINT;
END_VAR
pNode := __NEW(MUL_SINT);
Clone := pNode^;
END_METHOD

METHOD PROTECTED OnExecute
VAR
END_VAR
out.Value := in1.Value * in2.Value;
END_METHOD

END_FUNCTION_BLOCK

// Core/Nodes/MUL/MUL_UDINT
{attribute 'linkalways'} 
{attribute 'no_explicit_call' := 'This FB is a CLASS and must be accessed using methods or properties'}
{attribute 'enable_dynamic_creation'}
FUNCTION_BLOCK FINAL MUL_UDINT EXTENDS Node
VAR
	in1 : _UDINT(0);
	in2 : _UDINT(0);
	out : _UDINT(0);
END_VAR

METHOD FB_init : BOOL
VAR_INPUT
	bInitRetains : BOOL; // if TRUE, the retain variables are initialized (warm start / cold start)
	bInCopyCode : BOOL;  // if TRUE, the instance afterwards gets moved into the copy code (online change)
END_VAR
AddInput('in1',THIS^.in1);
AddInput('in2',THIS^.in2);
AddOutput('out', THIS^.out);
END_METHOD

METHOD PUBLIC Clone : I_Node
VAR
	pNode : POINTER TO MUL_UDINT;
END_VAR
pNode := __NEW(MUL_UDINT);
Clone := pNode^;
END_METHOD

METHOD PROTECTED OnExecute
VAR
END_VAR
out.Value := in1.Value * in2.Value;
END_METHOD

END_FUNCTION_BLOCK

// Core/Nodes/MUL/MUL_UINT
{attribute 'linkalways'} 
{attribute 'no_explicit_call' := 'This FB is a CLASS and must be accessed using methods or properties'}
{attribute 'enable_dynamic_creation'}
FUNCTION_BLOCK FINAL MUL_UINT EXTENDS Node
VAR
	in1 : _UINT(0);
	in2 : _UINT(0);
	out : _UINT(0);
END_VAR

METHOD FB_init : BOOL
VAR_INPUT
	bInitRetains : BOOL; // if TRUE, the retain variables are initialized (warm start / cold start)
	bInCopyCode : BOOL;  // if TRUE, the instance afterwards gets moved into the copy code (online change)
END_VAR
AddInput('in1',THIS^.in1);
AddInput('in2',THIS^.in2);
AddOutput('out', THIS^.out);
END_METHOD

METHOD PUBLIC Clone : I_Node
VAR
	pNode : POINTER TO MUL_UINT;
END_VAR
pNode := __NEW(MUL_UINT);
Clone := pNode^;
END_METHOD

METHOD PROTECTED OnExecute
VAR
END_VAR
out.Value := in1.Value * in2.Value;
END_METHOD

END_FUNCTION_BLOCK

// Core/Nodes/MUL/MUL_ULINT
{attribute 'linkalways'} 
{attribute 'no_explicit_call' := 'This FB is a CLASS and must be accessed using methods or properties'}
{attribute 'enable_dynamic_creation'}
FUNCTION_BLOCK FINAL MUL_ULINT EXTENDS Node
VAR
	in1 : _ULINT(0);
	in2 : _ULINT(0);
	out : _ULINT(0);
END_VAR

METHOD FB_init : BOOL
VAR_INPUT
	bInitRetains : BOOL; // if TRUE, the retain variables are initialized (warm start / cold start)
	bInCopyCode : BOOL;  // if TRUE, the instance afterwards gets moved into the copy code (online change)
END_VAR
AddInput('in1',THIS^.in1);
AddInput('in2',THIS^.in2);
AddOutput('out', THIS^.out);
END_METHOD

METHOD PUBLIC Clone : I_Node
VAR
	pNode : POINTER TO MUL_ULINT;
END_VAR
pNode := __NEW(MUL_ULINT);
Clone := pNode^;
END_METHOD

METHOD PROTECTED OnExecute
VAR
END_VAR
out.Value := in1.Value * in2.Value;
END_METHOD

END_FUNCTION_BLOCK

// Core/Nodes/MUL/MUL_USINT
{attribute 'linkalways'} 
{attribute 'no_explicit_call' := 'This FB is a CLASS and must be accessed using methods or properties'}
{attribute 'enable_dynamic_creation'}
FUNCTION_BLOCK FINAL MUL_USINT EXTENDS Node
VAR
	in1 : _USINT(0);
	in2 : _USINT(0);
	out : _USINT(0);
END_VAR

METHOD FB_init : BOOL
VAR_INPUT
	bInitRetains : BOOL; // if TRUE, the retain variables are initialized (warm start / cold start)
	bInCopyCode : BOOL;  // if TRUE, the instance afterwards gets moved into the copy code (online change)
END_VAR
AddInput('in1',THIS^.in1);
AddInput('in2',THIS^.in2);
AddOutput('out', THIS^.out);
END_METHOD

METHOD PUBLIC Clone : I_Node
VAR
	pNode : POINTER TO MUL_USINT;
END_VAR
pNode := __NEW(MUL_USINT);
Clone := pNode^;
END_METHOD

METHOD PROTECTED OnExecute
VAR
END_VAR
out.Value := in1.Value * in2.Value;
END_METHOD

END_FUNCTION_BLOCK

// Core/Nodes/MUL/MUL_WORD
{attribute 'linkalways'} 
{attribute 'no_explicit_call' := 'This FB is a CLASS and must be accessed using methods or properties'}
{attribute 'enable_dynamic_creation'}
FUNCTION_BLOCK FINAL MUL_WORD EXTENDS Node
VAR
	in1 : _WORD(0);
	in2 : _WORD(0);
	out : _WORD(0);
END_VAR

METHOD FB_init : BOOL
VAR_INPUT
	bInitRetains : BOOL; // if TRUE, the retain variables are initialized (warm start / cold start)
	bInCopyCode : BOOL;  // if TRUE, the instance afterwards gets moved into the copy code (online change)
END_VAR
AddInput('in1',THIS^.in1);
AddInput('in2',THIS^.in2);
AddOutput('out', THIS^.out);
END_METHOD

METHOD PUBLIC Clone : I_Node
VAR
	pNode : POINTER TO MUL_WORD;
END_VAR
pNode := __NEW(MUL_WORD);
Clone := pNode^;
END_METHOD

METHOD PROTECTED OnExecute
VAR
END_VAR
out.Value := in1.Value - in2.Value;
END_METHOD

END_FUNCTION_BLOCK

// Core/Nodes/SUB/SUB_BYTE
{attribute 'linkalways'} 
{attribute 'no_explicit_call' := 'This FB is a CLASS and must be accessed using methods or properties'}
{attribute 'enable_dynamic_creation'}
FUNCTION_BLOCK FINAL SUB_BYTE EXTENDS Node
VAR
	in1 : _BYTE(0);
	in2 : _BYTE(0);
	out : _BYTE(0);
END_VAR

METHOD FB_init : BOOL
VAR_INPUT
	bInitRetains : BOOL; // if TRUE, the retain variables are initialized (warm start / cold start)
	bInCopyCode : BOOL;  // if TRUE, the instance afterwards gets moved into the copy code (online change)
END_VAR
AddInput('in1',THIS^.in1);
AddInput('in2',THIS^.in2);
AddOutput('out', THIS^.out);
END_METHOD

METHOD PUBLIC Clone : I_Node
VAR
	pNode : POINTER TO SUB_BYTE;
END_VAR
pNode := __NEW(SUB_BYTE);
Clone := pNode^;
END_METHOD

METHOD PROTECTED OnExecute
VAR
END_VAR
out.Value := in1.Value - in2.Value;
END_METHOD

END_FUNCTION_BLOCK

// Core/Nodes/SUB/SUB_DINT
{attribute 'linkalways'} 
{attribute 'no_explicit_call' := 'This FB is a CLASS and must be accessed using methods or properties'}
{attribute 'enable_dynamic_creation'}
FUNCTION_BLOCK FINAL SUB_DINT EXTENDS Node
VAR
	in1 : _DINT(0);
	in2 : _DINT(0);
	out : _DINT(0);
END_VAR

METHOD FB_init : BOOL
VAR_INPUT
	bInitRetains : BOOL; // if TRUE, the retain variables are initialized (warm start / cold start)
	bInCopyCode : BOOL;  // if TRUE, the instance afterwards gets moved into the copy code (online change)
END_VAR
AddInput('in1',THIS^.in1);
AddInput('in2',THIS^.in2);
AddOutput('out', THIS^.out);
END_METHOD

METHOD PUBLIC Clone : I_Node
VAR
	pNode : POINTER TO SUB_DINT;
END_VAR
pNode := __NEW(SUB_DINT);
Clone := pNode^;
END_METHOD

METHOD PROTECTED OnExecute
VAR
END_VAR
out.Value := in1.Value - in2.Value;
END_METHOD

END_FUNCTION_BLOCK

// Core/Nodes/SUB/SUB_DWORD
{attribute 'linkalways'} 
{attribute 'no_explicit_call' := 'This FB is a CLASS and must be accessed using methods or properties'}
{attribute 'enable_dynamic_creation'}
FUNCTION_BLOCK FINAL SUB_DWORD EXTENDS Node
VAR
	in1 : _DWORD(0);
	in2 : _DWORD(0);
	out : _DWORD(0);
END_VAR

METHOD FB_init : BOOL
VAR_INPUT
	bInitRetains : BOOL; // if TRUE, the retain variables are initialized (warm start / cold start)
	bInCopyCode : BOOL;  // if TRUE, the instance afterwards gets moved into the copy code (online change)
END_VAR
AddInput('in1',THIS^.in1);
AddInput('in2',THIS^.in2);
AddOutput('out', THIS^.out);
END_METHOD

METHOD PUBLIC Clone : I_Node
VAR
	pNode : POINTER TO SUB_DWORD;
END_VAR
pNode := __NEW(SUB_DWORD);
Clone := pNode^;
END_METHOD

METHOD PROTECTED OnExecute
VAR
END_VAR
out.Value := in1.Value - in2.Value;
END_METHOD

END_FUNCTION_BLOCK

// Core/Nodes/SUB/SUB_INT
{attribute 'linkalways'} 
{attribute 'no_explicit_call' := 'This FB is a CLASS and must be accessed using methods or properties'}
{attribute 'enable_dynamic_creation'}
FUNCTION_BLOCK FINAL SUB_INT EXTENDS Node
VAR
	in1 : _INT(0);
	in2 : _INT(0);
	out : _INT(0);
END_VAR

METHOD FB_init : BOOL
VAR_INPUT
	bInitRetains : BOOL; // if TRUE, the retain variables are initialized (warm start / cold start)
	bInCopyCode : BOOL;  // if TRUE, the instance afterwards gets moved into the copy code (online change)
END_VAR
AddInput('in1',THIS^.in1);
AddInput('in2',THIS^.in2);
AddOutput('out', THIS^.out);
END_METHOD

METHOD PUBLIC Clone : I_Node
VAR
	pNode : POINTER TO SUB_INT;
END_VAR
pNode := __NEW(SUB_INT);
Clone := pNode^;
END_METHOD

METHOD PROTECTED OnExecute
VAR
END_VAR
out.Value := in1.Value - in2.Value;
END_METHOD

END_FUNCTION_BLOCK

// Core/Nodes/SUB/SUB_LINT
{attribute 'linkalways'} 
{attribute 'no_explicit_call' := 'This FB is a CLASS and must be accessed using methods or properties'}
{attribute 'enable_dynamic_creation'}
FUNCTION_BLOCK FINAL SUB_LINT EXTENDS Node
VAR
	in1 : _LINT(0);
	in2 : _LINT(0);
	out : _LINT(0);
END_VAR

METHOD FB_init : BOOL
VAR_INPUT
	bInitRetains : BOOL; // if TRUE, the retain variables are initialized (warm start / cold start)
	bInCopyCode : BOOL;  // if TRUE, the instance afterwards gets moved into the copy code (online change)
END_VAR
AddInput('in1',THIS^.in1);
AddInput('in2',THIS^.in2);
AddOutput('out', THIS^.out);
END_METHOD

METHOD PUBLIC Clone : I_Node
VAR
	pNode : POINTER TO SUB_LINT;
END_VAR
pNode := __NEW(SUB_LINT);
Clone := pNode^;
END_METHOD

METHOD PROTECTED OnExecute
VAR
END_VAR
out.Value := in1.Value - in2.Value;
END_METHOD

END_FUNCTION_BLOCK

// Core/Nodes/SUB/SUB_LREAL
{attribute 'linkalways'} 
{attribute 'no_explicit_call' := 'This FB is a CLASS and must be accessed using methods or properties'}
{attribute 'enable_dynamic_creation'}
FUNCTION_BLOCK FINAL SUB_LREAL EXTENDS Node
VAR
	in1 : _LREAL(0.0);
	in2 : _LREAL(0.0);
	out : _LREAL(0.0);
END_VAR

METHOD FB_init : BOOL
VAR_INPUT
	bInitRetains : BOOL; // if TRUE, the retain variables are initialized (warm start / cold start)
	bInCopyCode : BOOL;  // if TRUE, the instance afterwards gets moved into the copy code (online change)
END_VAR
AddInput('in1',THIS^.in1);
AddInput('in2',THIS^.in2);
AddOutput('out', THIS^.out);
END_METHOD

METHOD PUBLIC Clone : I_Node
VAR
	pNode : POINTER TO SUB_LREAL;
END_VAR
pNode := __NEW(SUB_LREAL);
Clone := pNode^;
END_METHOD

METHOD PROTECTED OnExecute
VAR
END_VAR
out.Value := in1.Value - in2.Value;
END_METHOD

END_FUNCTION_BLOCK

// Core/Nodes/SUB/SUB_LWORD
{attribute 'linkalways'} 
{attribute 'no_explicit_call' := 'This FB is a CLASS and must be accessed using methods or properties'}
{attribute 'enable_dynamic_creation'}
FUNCTION_BLOCK FINAL SUB_LWORD EXTENDS Node
VAR
	in1 : _LWORD(0);
	in2 : _LWORD(0);
	out : _LWORD(0);
END_VAR

METHOD FB_init : BOOL
VAR_INPUT
	bInitRetains : BOOL; // if TRUE, the retain variables are initialized (warm start / cold start)
	bInCopyCode : BOOL;  // if TRUE, the instance afterwards gets moved into the copy code (online change)
END_VAR
AddInput('in1',THIS^.in1);
AddInput('in2',THIS^.in2);
AddOutput('out', THIS^.out);
END_METHOD

METHOD PUBLIC Clone : I_Node
VAR
	pNode : POINTER TO SUB_LWORD;
END_VAR
pNode := __NEW(SUB_LWORD);
Clone := pNode^;
END_METHOD

METHOD PROTECTED OnExecute
VAR
END_VAR
out.Value := in1.Value - in2.Value;
END_METHOD

END_FUNCTION_BLOCK

// Core/Nodes/SUB/SUB_REAL
{attribute 'linkalways'} 
{attribute 'no_explicit_call' := 'This FB is a CLASS and must be accessed using methods or properties'}
{attribute 'enable_dynamic_creation'}
FUNCTION_BLOCK FINAL SUB_REAL EXTENDS Node
VAR
	in1 : _REAL(0.0);
	in2 : _REAL(0.0);
	out : _REAL(0.0);
END_VAR

METHOD FB_init : BOOL
VAR_INPUT
	bInitRetains : BOOL; // if TRUE, the retain variables are initialized (warm start / cold start)
	bInCopyCode : BOOL;  // if TRUE, the instance afterwards gets moved into the copy code (online change)
END_VAR
AddInput('in1',THIS^.in1);
AddInput('in2',THIS^.in2);
AddOutput('out', THIS^.out);
END_METHOD

METHOD PUBLIC Clone : I_Node
VAR
	pNode : POINTER TO SUB_REAL;
END_VAR
pNode := __NEW(SUB_REAL);
Clone := pNode^;
END_METHOD

METHOD PROTECTED OnExecute
VAR
END_VAR
out.Value := in1.Value - in2.Value;
END_METHOD

END_FUNCTION_BLOCK

// Core/Nodes/SUB/SUB_SINT
{attribute 'linkalways'} 
{attribute 'no_explicit_call' := 'This FB is a CLASS and must be accessed using methods or properties'}
{attribute 'enable_dynamic_creation'}
FUNCTION_BLOCK FINAL SUB_SINT EXTENDS Node
VAR
	in1 : _SINT(0);
	in2 : _SINT(0);
	out : _SINT(0);
END_VAR

METHOD FB_init : BOOL
VAR_INPUT
	bInitRetains : BOOL; // if TRUE, the retain variables are initialized (warm start / cold start)
	bInCopyCode : BOOL;  // if TRUE, the instance afterwards gets moved into the copy code (online change)
END_VAR
AddInput('in1',THIS^.in1);
AddInput('in2',THIS^.in2);
AddOutput('out', THIS^.out);
END_METHOD

METHOD PUBLIC Clone : I_Node
VAR
	pNode : POINTER TO SUB_SINT;
END_VAR
pNode := __NEW(SUB_SINT);
Clone := pNode^;
END_METHOD

METHOD PROTECTED OnExecute
VAR
END_VAR
out.Value := in1.Value - in2.Value;
END_METHOD

END_FUNCTION_BLOCK

// Core/Nodes/SUB/SUB_UDINT
{attribute 'linkalways'} 
{attribute 'no_explicit_call' := 'This FB is a CLASS and must be accessed using methods or properties'}
{attribute 'enable_dynamic_creation'}
FUNCTION_BLOCK FINAL SUB_UDINT EXTENDS Node
VAR
	in1 : _UDINT(0);
	in2 : _UDINT(0);
	out : _UDINT(0);
END_VAR

METHOD FB_init : BOOL
VAR_INPUT
	bInitRetains : BOOL; // if TRUE, the retain variables are initialized (warm start / cold start)
	bInCopyCode : BOOL;  // if TRUE, the instance afterwards gets moved into the copy code (online change)
END_VAR
AddInput('in1',THIS^.in1);
AddInput('in2',THIS^.in2);
AddOutput('out', THIS^.out);
END_METHOD

METHOD PUBLIC Clone : I_Node
VAR
	pNode : POINTER TO SUB_UDINT;
END_VAR
pNode := __NEW(SUB_UDINT);
Clone := pNode^;
END_METHOD

METHOD PROTECTED OnExecute
VAR
END_VAR
out.Value := in1.Value - in2.Value;
END_METHOD

END_FUNCTION_BLOCK

// Core/Nodes/SUB/SUB_UINT
{attribute 'linkalways'} 
{attribute 'no_explicit_call' := 'This FB is a CLASS and must be accessed using methods or properties'}
{attribute 'enable_dynamic_creation'}
FUNCTION_BLOCK FINAL SUB_UINT EXTENDS Node
VAR
	in1 : _UINT(0);
	in2 : _UINT(0);
	out : _UINT(0);
END_VAR

METHOD FB_init : BOOL
VAR_INPUT
	bInitRetains : BOOL; // if TRUE, the retain variables are initialized (warm start / cold start)
	bInCopyCode : BOOL;  // if TRUE, the instance afterwards gets moved into the copy code (online change)
END_VAR
AddInput('in1',THIS^.in1);
AddInput('in2',THIS^.in2);
AddOutput('out', THIS^.out);
END_METHOD

METHOD PUBLIC Clone : I_Node
VAR
	pNode : POINTER TO SUB_UINT;
END_VAR
pNode := __NEW(SUB_UINT);
Clone := pNode^;
END_METHOD

METHOD PROTECTED OnExecute
VAR
END_VAR
out.Value := in1.Value - in2.Value;
END_METHOD

END_FUNCTION_BLOCK

// Core/Nodes/SUB/SUB_ULINT
{attribute 'linkalways'} 
{attribute 'no_explicit_call' := 'This FB is a CLASS and must be accessed using methods or properties'}
{attribute 'enable_dynamic_creation'}
FUNCTION_BLOCK FINAL SUB_ULINT EXTENDS Node
VAR
	in1 : _ULINT(0);
	in2 : _ULINT(0);
	out : _ULINT(0);
END_VAR

METHOD FB_init : BOOL
VAR_INPUT
	bInitRetains : BOOL; // if TRUE, the retain variables are initialized (warm start / cold start)
	bInCopyCode : BOOL;  // if TRUE, the instance afterwards gets moved into the copy code (online change)
END_VAR
AddInput('in1',THIS^.in1);
AddInput('in2',THIS^.in2);
AddOutput('out', THIS^.out);
END_METHOD

METHOD PUBLIC Clone : I_Node
VAR
	pNode : POINTER TO SUB_ULINT;
END_VAR
pNode := __NEW(SUB_ULINT);
Clone := pNode^;
END_METHOD

METHOD PROTECTED OnExecute
VAR
END_VAR
out.Value := in1.Value - in2.Value;
END_METHOD

END_FUNCTION_BLOCK

// Core/Nodes/SUB/SUB_USINT
{attribute 'linkalways'} 
{attribute 'no_explicit_call' := 'This FB is a CLASS and must be accessed using methods or properties'}
{attribute 'enable_dynamic_creation'}
FUNCTION_BLOCK FINAL SUB_USINT EXTENDS Node
VAR
	in1 : _USINT(0);
	in2 : _USINT(0);
	out : _USINT(0);
END_VAR

METHOD FB_init : BOOL
VAR_INPUT
	bInitRetains : BOOL; // if TRUE, the retain variables are initialized (warm start / cold start)
	bInCopyCode : BOOL;  // if TRUE, the instance afterwards gets moved into the copy code (online change)
END_VAR
AddInput('in1',THIS^.in1);
AddInput('in2',THIS^.in2);
AddOutput('out', THIS^.out);
END_METHOD

METHOD PUBLIC Clone : I_Node
VAR
	pNode : POINTER TO SUB_USINT;
END_VAR
pNode := __NEW(SUB_USINT);
Clone := pNode^;
END_METHOD

METHOD PROTECTED OnExecute
VAR
END_VAR
out.Value := in1.Value - in2.Value;
END_METHOD

END_FUNCTION_BLOCK

// Core/Nodes/SUB/SUB_WORD
{attribute 'linkalways'} 
{attribute 'no_explicit_call' := 'This FB is a CLASS and must be accessed using methods or properties'}
{attribute 'enable_dynamic_creation'}
FUNCTION_BLOCK FINAL SUB_WORD EXTENDS Node
VAR
	in1 : _WORD(0);
	in2 : _WORD(0);
	out : _WORD(0);
END_VAR

METHOD FB_init : BOOL
VAR_INPUT
	bInitRetains : BOOL; // if TRUE, the retain variables are initialized (warm start / cold start)
	bInCopyCode : BOOL;  // if TRUE, the instance afterwards gets moved into the copy code (online change)
END_VAR
AddInput('in1',THIS^.in1);
AddInput('in2',THIS^.in2);
AddOutput('out', THIS^.out);
END_METHOD

METHOD PUBLIC Clone : I_Node
VAR
	pNode : POINTER TO SUB_WORD;
END_VAR
pNode := __NEW(SUB_WORD);
Clone := pNode^;
END_METHOD

METHOD PROTECTED OnExecute
VAR
END_VAR
out.Value := in1.Value - in2.Value;
END_METHOD

END_FUNCTION_BLOCK

// Core/MathCorePack
{attribute 'linkalways'} 
{attribute 'no_explicit_call' := 'This FB is a CLASS and must be accessed using methods or properties'}
{attribute 'enable_dynamic_creation'}
FUNCTION_BLOCK MathCorePack IMPLEMENTS I_GraphPack
VAR
	ADD_BYTE : ADD_BYTE;
	ADD_DINT : ADD_DINT;
	ADD_DWORD : ADD_DWORD;
	ADD_INT : ADD_INT;
	ADD_LINT : ADD_LINT;
	ADD_LREAL : ADD_LREAL;
	ADD_LWORD : ADD_LWORD;
	ADD_REAL : ADD_REAL;
	ADD_SINT : ADD_SINT;
	ADD_UDINT : ADD_UDINT;
	ADD_UINT : ADD_UINT;
	ADD_ULINT : ADD_ULINT;
	ADD_USINT : ADD_USINT;
	ADD_WORD : ADD_WORD;
	
	SUB_BYTE : SUB_BYTE;
	SUB_DINT : SUB_DINT;
	SUB_DWORD : SUB_DWORD;
	SUB_INT : SUB_INT;
	SUB_LINT : SUB_LINT;
	SUB_LREAL : SUB_LREAL;
	SUB_LWORD : SUB_LWORD;
	SUB_REAL : SUB_REAL;
	SUB_SINT : SUB_SINT;
	SUB_UDINT : SUB_UDINT;
	SUB_UINT : SUB_UINT;
	SUB_ULINT : SUB_ULINT;
	SUB_USINT : SUB_USINT;
	SUB_WORD : SUB_WORD;
	
	MUL_BYTE : MUL_BYTE;
	MUL_DINT : MUL_DINT;
	MUL_DWORD : MUL_DWORD;
	MUL_INT : MUL_INT;
	MUL_LINT : MUL_LINT;
	MUL_LREAL : MUL_LREAL;
	MUL_LWORD : MUL_LWORD;
	MUL_REAL : MUL_REAL;
	MUL_SINT : MUL_SINT;
	MUL_UDINT : MUL_UDINT;
	MUL_UINT : MUL_UINT;
	MUL_ULINT : MUL_ULINT;
	MUL_USINT : MUL_USINT;
	MUL_WORD : MUL_WORD;
	
	DIV_BYTE : DIV_BYTE;
	DIV_DINT : DIV_DINT;
	DIV_DWORD : DIV_DWORD;
	DIV_INT : DIV_INT;
	DIV_LINT : DIV_LINT;
	DIV_LREAL : DIV_LREAL;
	DIV_LWORD : DIV_LWORD;
	DIV_REAL : DIV_REAL;
	DIV_SINT : DIV_SINT;
	DIV_UDINT : DIV_UDINT;
	DIV_UINT : DIV_UINT;
	DIV_ULINT : DIV_ULINT;
	DIV_USINT : DIV_USINT;
	DIV_WORD : DIV_WORD;
	
	MOD_BYTE : MOD_BYTE;
	MOD_DINT : MOD_DINT;
	MOD_DWORD : MOD_DWORD;
	MOD_INT : MOD_INT;
	MOD_LINT : MOD_LINT;
	MOD_LREAL : MOD_LREAL;
	MOD_LWORD : MOD_LWORD;
	MOD_SINT : MOD_SINT;
	MOD_UDINT : MOD_UDINT;
	MOD_UINT : MOD_UINT;
	MOD_ULINT : MOD_ULINT;
	MOD_USINT : MOD_USINT;
	MOD_WORD : MOD_WORD;
	

END_VAR

METHOD Register
VAR_INPUT
	Datatypes : I_Datatypes;
	NodeFactory : I_NodeFactory;
END_VAR
NodeFactory.AddNodeAsPrototype('Math/Core/ADD/ADD_BYTE',ADD_BYTE);
NodeFactory.AddNodeAsPrototype('Math/Core/ADD/ADD_DINT',ADD_DINT);
NodeFactory.AddNodeAsPrototype('Math/Core/ADD/ADD_DWORD',ADD_DWORD);
NodeFactory.AddNodeAsPrototype('Math/Core/ADD/ADD_INT',ADD_INT);
NodeFactory.AddNodeAsPrototype('Math/Core/ADD/ADD_LINT',ADD_LINT);
NodeFactory.AddNodeAsPrototype('Math/Core/ADD/ADD_LREAL',ADD_LREAL);
NodeFactory.AddNodeAsPrototype('Math/Core/ADD/ADD_LWORD',ADD_LWORD);
NodeFactory.AddNodeAsPrototype('Math/Core/ADD/ADD_REAL',ADD_REAL);
NodeFactory.AddNodeAsPrototype('Math/Core/ADD/ADD_SINT',ADD_SINT);
NodeFactory.AddNodeAsPrototype('Math/Core/ADD/ADD_UDINT',ADD_UDINT);
NodeFactory.AddNodeAsPrototype('Math/Core/ADD/ADD_UINT',ADD_UINT);
NodeFactory.AddNodeAsPrototype('Math/Core/ADD/ADD_ULINT',ADD_ULINT);
NodeFactory.AddNodeAsPrototype('Math/Core/ADD/ADD_USINT',ADD_USINT);
NodeFactory.AddNodeAsPrototype('Math/Core/ADD/ADD_WORD',ADD_WORD);

NodeFactory.AddNodeAsPrototype('Math/Core/SUB/SUB_BYTE',SUB_BYTE);
NodeFactory.AddNodeAsPrototype('Math/Core/SUB/SUB_DINT',SUB_DINT);
NodeFactory.AddNodeAsPrototype('Math/Core/SUB/SUB_DWORD',SUB_DWORD);
NodeFactory.AddNodeAsPrototype('Math/Core/SUB/SUB_INT',SUB_INT);
NodeFactory.AddNodeAsPrototype('Math/Core/SUB/SUB_LINT',SUB_LINT);
NodeFactory.AddNodeAsPrototype('Math/Core/SUB/SUB_LREAL',SUB_LREAL);
NodeFactory.AddNodeAsPrototype('Math/Core/SUB/SUB_LWORD',SUB_LWORD);
NodeFactory.AddNodeAsPrototype('Math/Core/SUB/SUB_REAL',SUB_REAL);
NodeFactory.AddNodeAsPrototype('Math/Core/SUB/SUB_SINT',SUB_SINT);
NodeFactory.AddNodeAsPrototype('Math/Core/SUB/SUB_UDINT',SUB_UDINT);
NodeFactory.AddNodeAsPrototype('Math/Core/SUB/SUB_UINT',SUB_UINT);
NodeFactory.AddNodeAsPrototype('Math/Core/SUB/SUB_ULINT',SUB_ULINT);
NodeFactory.AddNodeAsPrototype('Math/Core/SUB/SUB_USINT',SUB_USINT);
NodeFactory.AddNodeAsPrototype('Math/Core/SUB/SUB_WORD',SUB_WORD);

NodeFactory.AddNodeAsPrototype('Math/Core/MUL/MUL_BYTE',MUL_BYTE);
NodeFactory.AddNodeAsPrototype('Math/Core/MUL/MUL_DINT',MUL_DINT);
NodeFactory.AddNodeAsPrototype('Math/Core/MUL/MUL_DWORD',MUL_DWORD);
NodeFactory.AddNodeAsPrototype('Math/Core/MUL/MUL_INT',MUL_INT);
NodeFactory.AddNodeAsPrototype('Math/Core/MUL/MUL_LINT',MUL_LINT);
NodeFactory.AddNodeAsPrototype('Math/Core/MUL/MUL_LREAL',MUL_LREAL);
NodeFactory.AddNodeAsPrototype('Math/Core/MUL/MUL_LWORD',MUL_LWORD);
NodeFactory.AddNodeAsPrototype('Math/Core/MUL/MUL_REAL',MUL_REAL);
NodeFactory.AddNodeAsPrototype('Math/Core/MUL/MUL_SINT',MUL_SINT);
NodeFactory.AddNodeAsPrototype('Math/Core/MUL/MUL_UDINT',MUL_UDINT);
NodeFactory.AddNodeAsPrototype('Math/Core/MUL/MUL_UINT',MUL_UINT);
NodeFactory.AddNodeAsPrototype('Math/Core/MUL/MUL_ULINT',MUL_ULINT);
NodeFactory.AddNodeAsPrototype('Math/Core/MUL/MUL_USINT',MUL_USINT);
NodeFactory.AddNodeAsPrototype('Math/Core/MUL/MUL_WORD',MUL_WORD);

NodeFactory.AddNodeAsPrototype('Math/Core/DIV/DIV_BYTE',DIV_BYTE);
NodeFactory.AddNodeAsPrototype('Math/Core/DIV/DIV_DINT',DIV_DINT);
NodeFactory.AddNodeAsPrototype('Math/Core/DIV/DIV_DWORD',DIV_DWORD);
NodeFactory.AddNodeAsPrototype('Math/Core/DIV/DIV_INT',DIV_INT);
NodeFactory.AddNodeAsPrototype('Math/Core/DIV/DIV_LINT',DIV_LINT);
NodeFactory.AddNodeAsPrototype('Math/Core/DIV/DIV_LREAL',DIV_LREAL);
NodeFactory.AddNodeAsPrototype('Math/Core/DIV/DIV_LWORD',DIV_LWORD);
NodeFactory.AddNodeAsPrototype('Math/Core/DIV/DIV_REAL',DIV_REAL);
NodeFactory.AddNodeAsPrototype('Math/Core/DIV/DIV_SINT',DIV_SINT);
NodeFactory.AddNodeAsPrototype('Math/Core/DIV/DIV_UDINT',DIV_UDINT);
NodeFactory.AddNodeAsPrototype('Math/Core/DIV/DIV_UINT',DIV_UINT);
NodeFactory.AddNodeAsPrototype('Math/Core/DIV/DIV_ULINT',DIV_ULINT);
NodeFactory.AddNodeAsPrototype('Math/Core/DIV/DIV_USINT',DIV_USINT);
NodeFactory.AddNodeAsPrototype('Math/Core/DIV/DIV_WORD',DIV_WORD);

NodeFactory.AddNodeAsPrototype('Math/Core/MOD/MOD_BYTE',MOD_BYTE);
NodeFactory.AddNodeAsPrototype('Math/Core/MOD/MOD_DINT',MOD_DINT);
NodeFactory.AddNodeAsPrototype('Math/Core/MOD/MOD_DWORD',MOD_DWORD);
NodeFactory.AddNodeAsPrototype('Math/Core/MOD/MOD_INT',MOD_INT);
NodeFactory.AddNodeAsPrototype('Math/Core/MOD/MOD_LINT',MOD_LINT);
NodeFactory.AddNodeAsPrototype('Math/Core/MOD/MOD_LREAL',MOD_LREAL);
NodeFactory.AddNodeAsPrototype('Math/Core/MOD/MOD_LWORD',MOD_LWORD);
NodeFactory.AddNodeAsPrototype('Math/Core/MOD/MOD_SINT',MOD_SINT);
NodeFactory.AddNodeAsPrototype('Math/Core/MOD/MOD_UDINT',MOD_UDINT);
NodeFactory.AddNodeAsPrototype('Math/Core/MOD/MOD_UINT',MOD_UINT);
NodeFactory.AddNodeAsPrototype('Math/Core/MOD/MOD_ULINT',MOD_ULINT);
NodeFactory.AddNodeAsPrototype('Math/Core/MOD/MOD_USINT',MOD_USINT);
NodeFactory.AddNodeAsPrototype('Math/Core/MOD/MOD_WORD',MOD_WORD);
END_METHOD

END_FUNCTION_BLOCK

// Logic/Nodes/AND/AND_BOOL
{attribute 'linkalways'} 
{attribute 'no_explicit_call' := 'This FB is a CLASS and must be accessed using methods or properties'}
{attribute 'enable_dynamic_creation'}
FUNCTION_BLOCK FINAL AND_BOOL EXTENDS Node
VAR
	in1 : _BOOL(FALSE);
	in2 : _BOOL(FALSE);
	out : _BOOL(FALSE);
END_VAR

METHOD FB_init : BOOL
VAR_INPUT
	bInitRetains : BOOL; // if TRUE, the retain variables are initialized (warm start / cold start)
	bInCopyCode : BOOL;  // if TRUE, the instance afterwards gets moved into the copy code (online change)
END_VAR
AddInput('in1',THIS^.in1);
AddInput('in2',THIS^.in2);
AddOutput('out', THIS^.out);
END_METHOD

METHOD PUBLIC Clone : I_Node
VAR
	pNode : POINTER TO AND_BOOL;
END_VAR
pNode := __NEW(AND_BOOL);
Clone := pNode^;
END_METHOD

METHOD PROTECTED OnExecute
VAR
END_VAR
out.Value := in1.Value AND in2.Value;
END_METHOD

END_FUNCTION_BLOCK

// Logic/Nodes/AND/AND_BYTE
{attribute 'linkalways'} 
{attribute 'no_explicit_call' := 'This FB is a CLASS and must be accessed using methods or properties'}
{attribute 'enable_dynamic_creation'}
FUNCTION_BLOCK FINAL AND_BYTE EXTENDS Node
VAR
	in1 : _BYTE(0);
	in2 : _BYTE(0);
	out : _BYTE(0);
END_VAR

METHOD FB_init : BOOL
VAR_INPUT
	bInitRetains : BOOL; // if TRUE, the retain variables are initialized (warm start / cold start)
	bInCopyCode : BOOL;  // if TRUE, the instance afterwards gets moved into the copy code (online change)
END_VAR
AddInput('in1',THIS^.in1);
AddInput('in2',THIS^.in2);
AddOutput('out', THIS^.out);
END_METHOD

METHOD PUBLIC Clone : I_Node
VAR
	pNode : POINTER TO AND_BYTE;
END_VAR
pNode := __NEW(AND_BYTE);
Clone := pNode^;
END_METHOD

